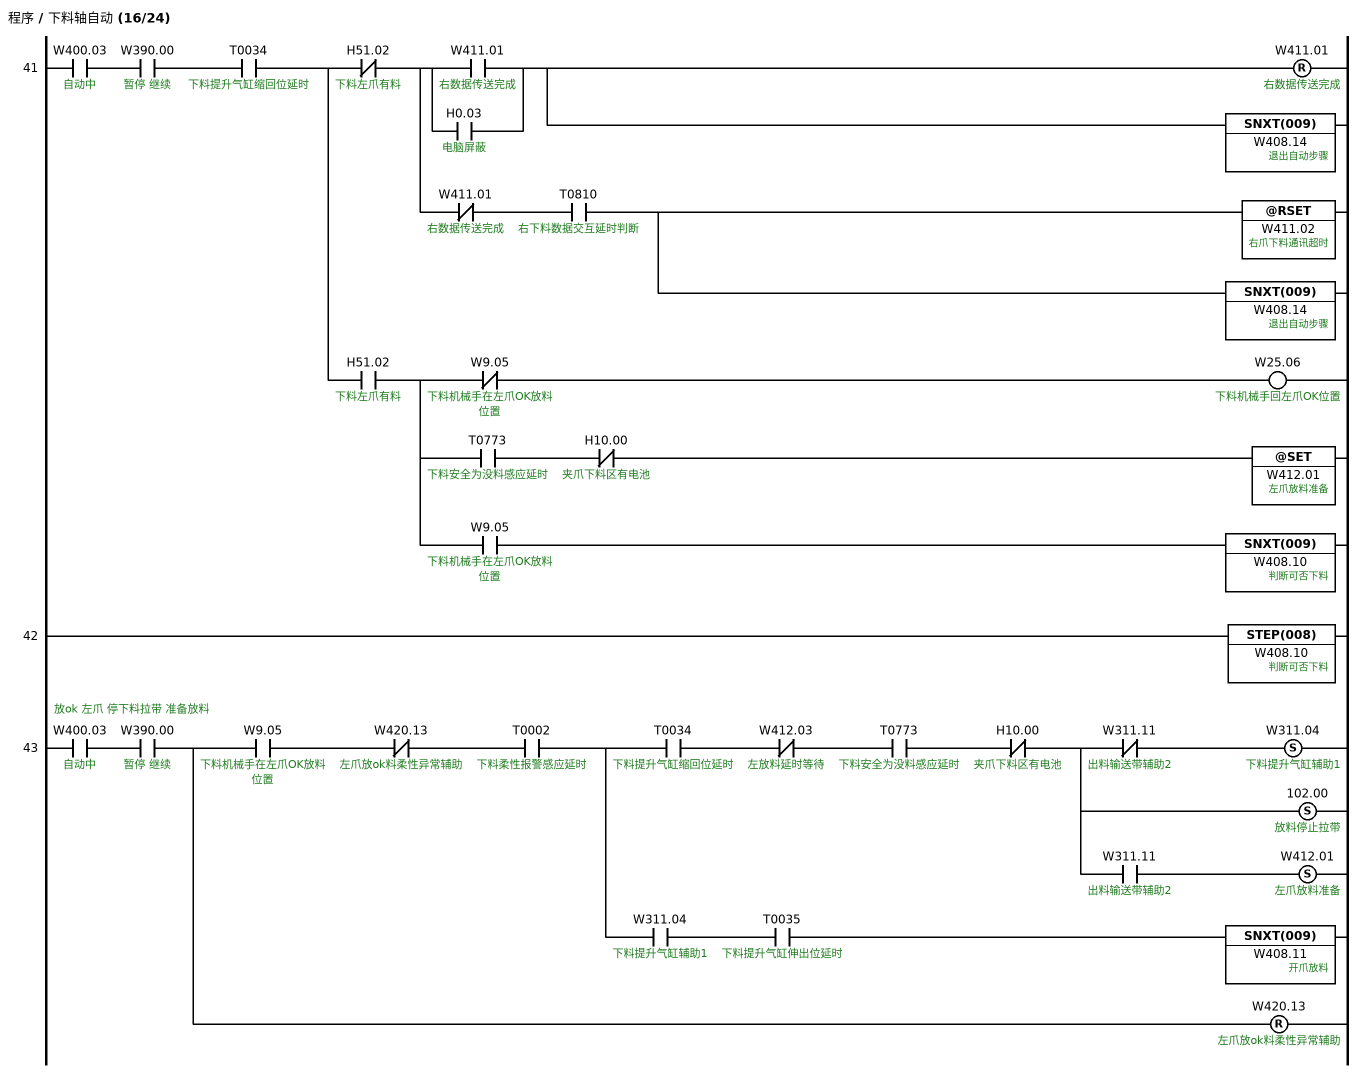
; rung 41
LD W400.03  ; 自动中
AND W390.00  ; 暂停 继续
AND T0034  ; 下料提升气缸缩回位延时
OUT TR0
ANDNOT H51.02  ; 下料左爪有料
OUT TR1
LD W411.01  ; 右数据传送完成
OR H0.03  ; 电脑屏蔽
ANDLD
RSET W411.01  ; 右数据传送完成
SNXT(009) W408.14  ; 退出自动步骤
LD TR1
ANDNOT W411.01  ; 右数据传送完成
AND T0810  ; 右下料数据交互延时判断
@RSET W411.02  ; 右爪下料通讯超时
SNXT(009) W408.14  ; 退出自动步骤
LD TR0
AND H51.02  ; 下料左爪有料
OUT TR0
ANDNOT W9.05  ; 下料机械手在左爪OK放料位置
OUT W25.06  ; 下料机械手回左爪OK位置
LD TR0
AND T0773  ; 下料安全为没料感应延时
ANDNOT H10.00  ; 夹爪下料区有电池
@SET W412.01  ; 左爪放料准备
LD TR0
AND W9.05  ; 下料机械手在左爪OK放料位置
SNXT(009) W408.10  ; 判断可否下料
; rung 42
STEP(008) W408.10  ; 判断可否下料
; rung 43: 放ok 左爪 停下料拉带 准备放料
LD W400.03  ; 自动中
AND W390.00  ; 暂停 继续
OUT TR0
AND W9.05  ; 下料机械手在左爪OK放料位置
ANDNOT W420.13  ; 左爪放ok料柔性异常辅助
AND T0002  ; 下料柔性报警感应延时
OUT TR1
AND T0034  ; 下料提升气缸缩回位延时
ANDNOT W412.03  ; 左放料延时等待
AND T0773  ; 下料安全为没料感应延时
ANDNOT H10.00  ; 夹爪下料区有电池
OUT TR2
ANDNOT W311.11  ; 出料输送带辅助2
SET W311.04  ; 下料提升气缸辅助1
LD TR2
SET 102.00  ; 放料停止拉带
AND W311.11  ; 出料输送带辅助2
SET W412.01  ; 左爪放料准备
LD TR1
AND W311.04  ; 下料提升气缸辅助1
AND T0035  ; 下料提升气缸伸出位延时
SNXT(009) W408.11  ; 开爪放料
LD TR0
RSET W420.13  ; 左爪放ok料柔性异常辅助

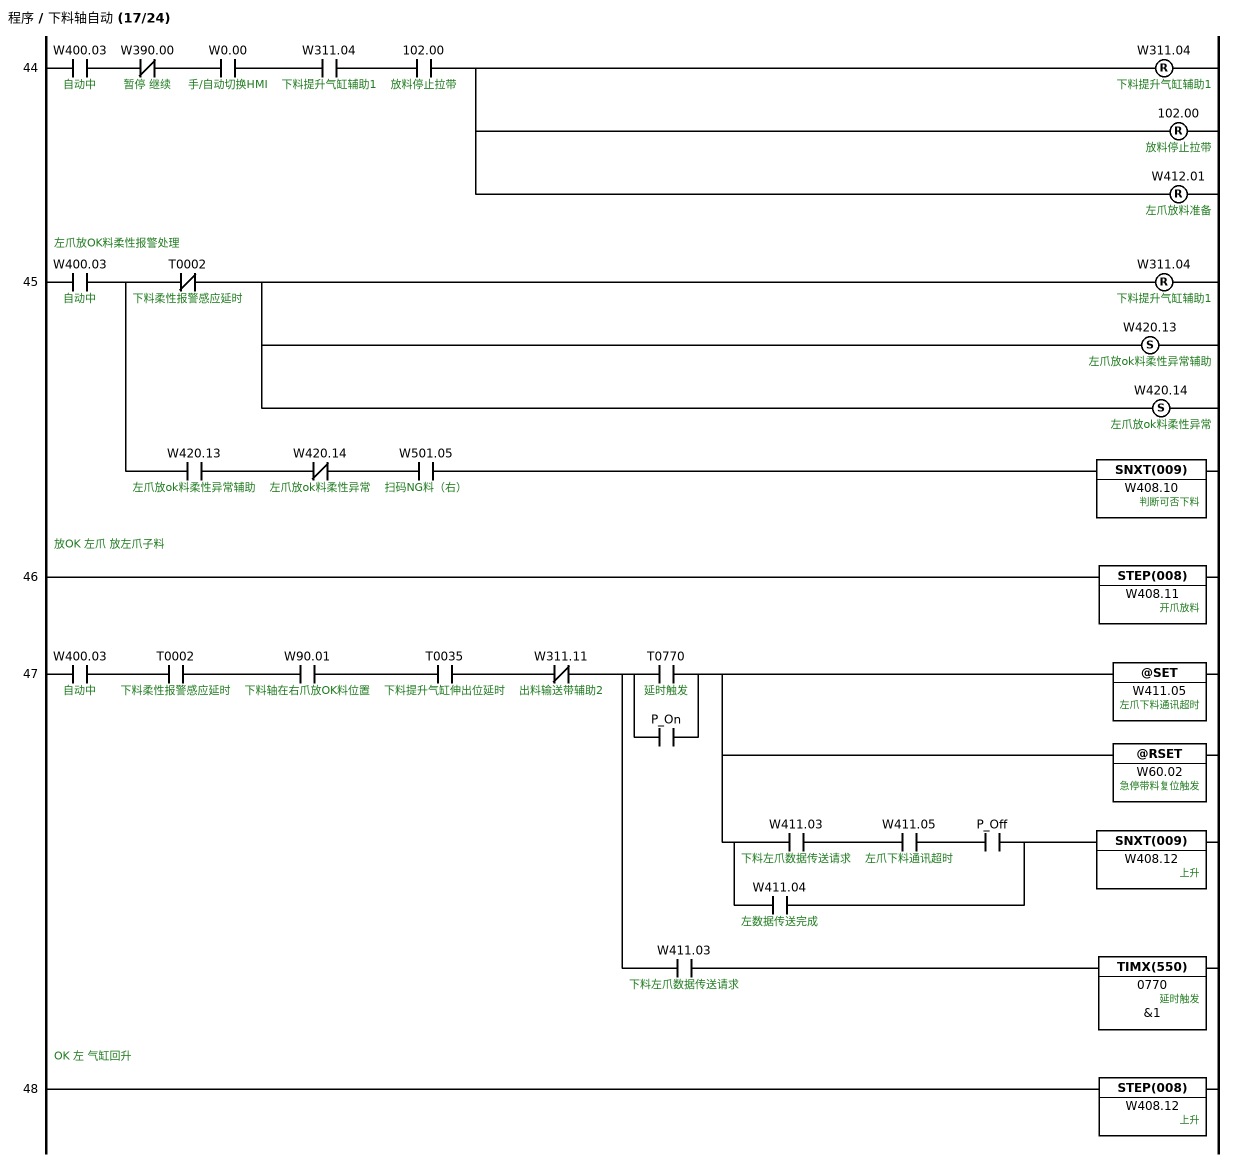
; rung 44
LD W400.03  ; 自动中
ANDNOT W390.00  ; 暂停 继续
AND W0.00  ; 手/自动切换HMI
AND W311.04  ; 下料提升气缸辅助1
AND 102.00  ; 放料停止拉带
RSET W311.04  ; 下料提升气缸辅助1
RSET 102.00  ; 放料停止拉带
RSET W412.01  ; 左爪放料准备
; rung 45: 左爪放OK料柔性报警处理
LD W400.03  ; 自动中
OUT TR0
ANDNOT T0002  ; 下料柔性报警感应延时
RSET W311.04  ; 下料提升气缸辅助1
SET W420.13  ; 左爪放ok料柔性异常辅助
SET W420.14  ; 左爪放ok料柔性异常
LD TR0
AND W420.13  ; 左爪放ok料柔性异常辅助
ANDNOT W420.14  ; 左爪放ok料柔性异常
AND W501.05  ; 扫码NG料（右）
SNXT(009) W408.10  ; 判断可否下料
; rung 46: 放OK 左爪 放左爪子料
STEP(008) W408.11  ; 开爪放料
; rung 47
LD W400.03  ; 自动中
AND T0002  ; 下料柔性报警感应延时
AND W90.01  ; 下料轴在右爪放OK料位置
AND T0035  ; 下料提升气缸伸出位延时
ANDNOT W311.11  ; 出料输送带辅助2
OUT TR0
LD T0770  ; 延时触发
OR P_On
ANDLD
@SET W411.05  ; 左爪下料通讯超时
@RSET W60.02  ; 急停带料复位触发
LD W411.03  ; 下料左爪数据传送请求
AND W411.05  ; 左爪下料通讯超时
AND P_Off
OR W411.04  ; 左数据传送完成
ANDLD
SNXT(009) W408.12  ; 上升
LD TR0
AND W411.03  ; 下料左爪数据传送请求
TIMX(550) 0770 &1  ; 延时触发
; rung 48: OK 左 气缸回升
STEP(008) W408.12  ; 上升

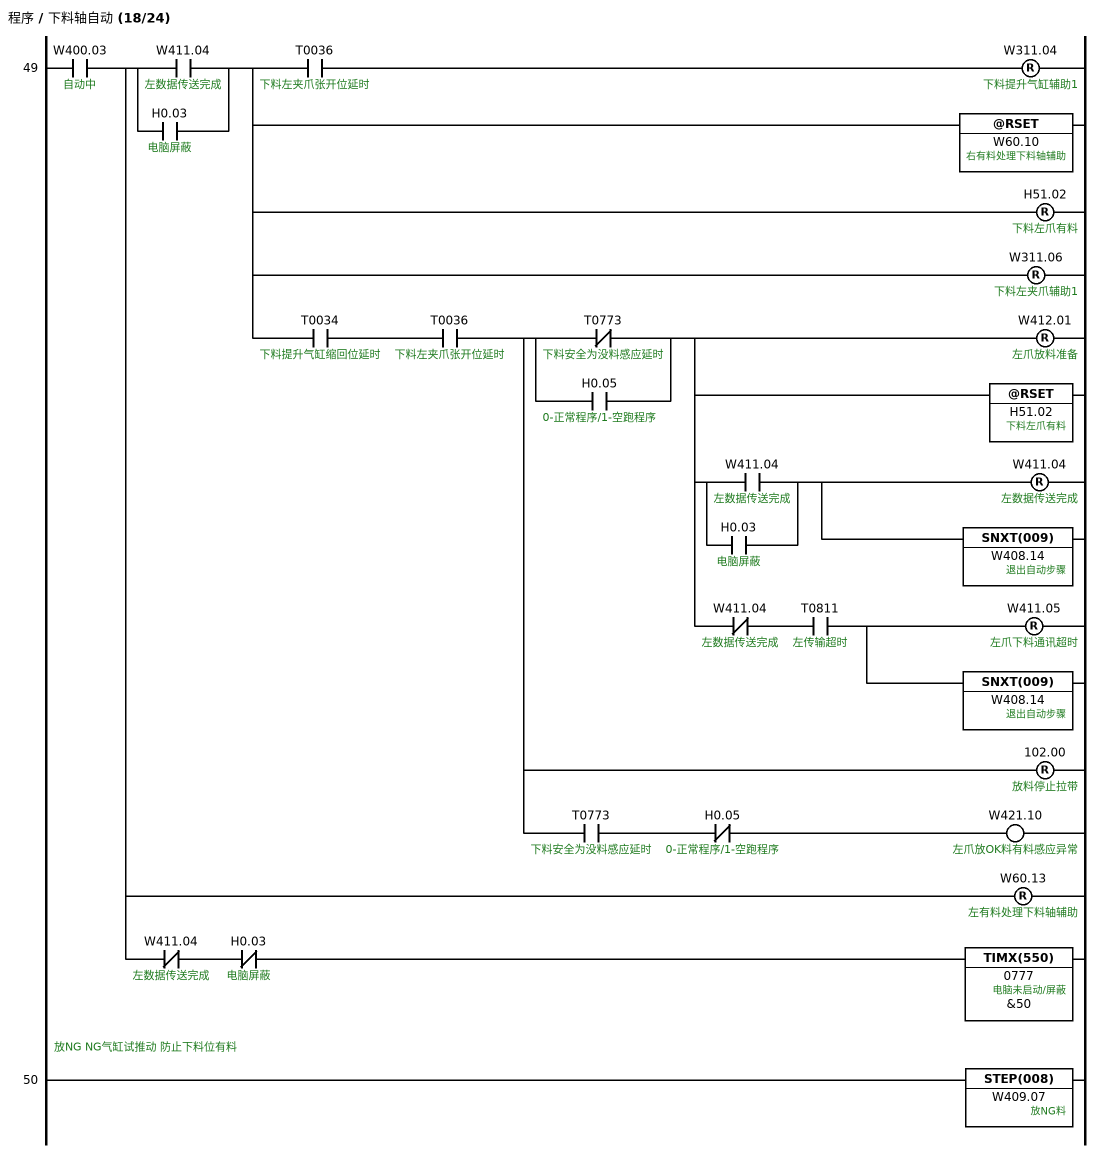
; rung 49
LD W400.03  ; 自动中
OUT TR0
LD W411.04  ; 左数据传送完成
OR H0.03  ; 电脑屏蔽
ANDLD
OUT TR1
AND T0036  ; 下料左夹爪张开位延时
RSET W311.04  ; 下料提升气缸辅助1
LD TR1
@RSET W60.10  ; 右有料处理下料轴辅助
RSET H51.02  ; 下料左爪有料
RSET W311.06  ; 下料左夹爪辅助1
AND T0034  ; 下料提升气缸缩回位延时
AND T0036  ; 下料左夹爪张开位延时
OUT TR1
LDNOT T0773  ; 下料安全为没料感应延时
OR H0.05  ; 0-正常程序/1-空跑程序
ANDLD
OUT TR2
RSET W412.01  ; 左爪放料准备
@RSET H51.02  ; 下料左爪有料
LD W411.04  ; 左数据传送完成
OR H0.03  ; 电脑屏蔽
ANDLD
RSET W411.04  ; 左数据传送完成
SNXT(009) W408.14  ; 退出自动步骤
LD TR2
ANDNOT W411.04  ; 左数据传送完成
AND T0811  ; 左传输超时
RSET W411.05  ; 左爪下料通讯超时
SNXT(009) W408.14  ; 退出自动步骤
LD TR1
RSET 102.00  ; 放料停止拉带
AND T0773  ; 下料安全为没料感应延时
ANDNOT H0.05  ; 0-正常程序/1-空跑程序
OUT W421.10  ; 左爪放OK料有料感应异常
LD TR0
RSET W60.13  ; 左有料处理下料轴辅助
ANDNOT W411.04  ; 左数据传送完成
ANDNOT H0.03  ; 电脑屏蔽
TIMX(550) 0777 &50  ; 电脑未启动/屏蔽
; rung 50: 放NG NG气缸试推动 防止下料位有料
STEP(008) W409.07  ; 放NG料

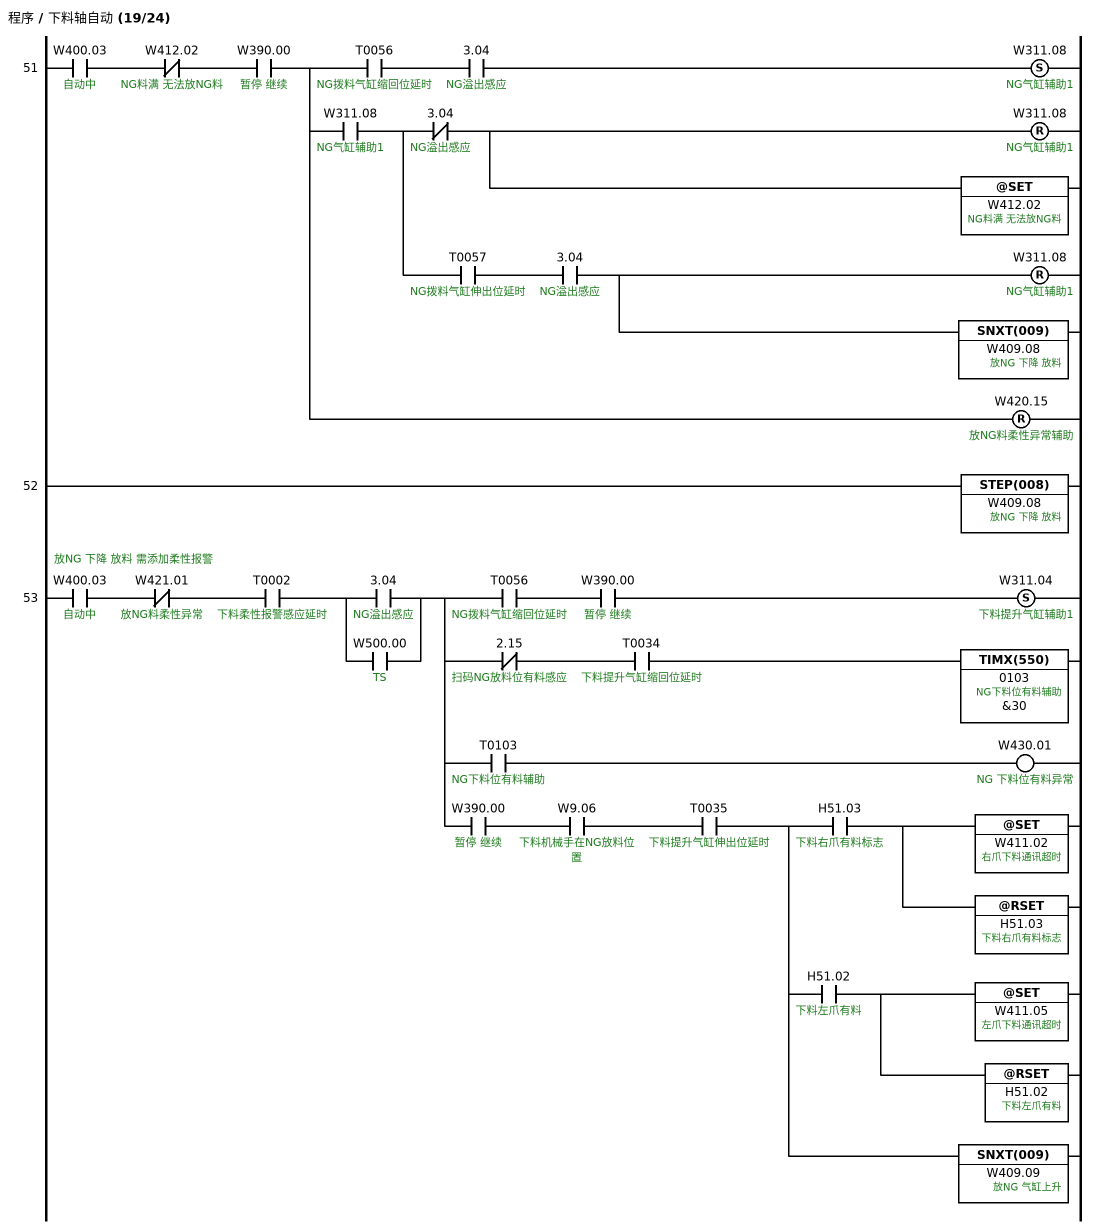
; rung 51
LD W400.03  ; 自动中
ANDNOT W412.02  ; NG料满 无法放NG料
AND W390.00  ; 暂停 继续
OUT TR0
AND T0056  ; NG拨料气缸缩回位延时
AND 3.04  ; NG溢出感应
SET W311.08  ; NG气缸辅助1
LD TR0
AND W311.08  ; NG气缸辅助1
OUT TR1
ANDNOT 3.04  ; NG溢出感应
RSET W311.08  ; NG气缸辅助1
@SET W412.02  ; NG料满 无法放NG料
LD TR1
AND T0057  ; NG拨料气缸伸出位延时
AND 3.04  ; NG溢出感应
RSET W311.08  ; NG气缸辅助1
SNXT(009) W409.08  ; 放NG 下降 放料
LD TR0
RSET W420.15  ; 放NG料柔性异常辅助
; rung 52
STEP(008) W409.08  ; 放NG 下降 放料
; rung 53: 放NG 下降 放料 需添加柔性报警
LD W400.03  ; 自动中
ANDNOT W421.01  ; 放NG料柔性异常
AND T0002  ; 下料柔性报警感应延时
LD 3.04  ; NG溢出感应
OR W500.00  ; TS
ANDLD
OUT TR0
AND T0056  ; NG拨料气缸缩回位延时
AND W390.00  ; 暂停 继续
SET W311.04  ; 下料提升气缸辅助1
LD TR0
ANDNOT 2.15  ; 扫码NG放料位有料感应
AND T0034  ; 下料提升气缸缩回位延时
TIMX(550) 0103 &30  ; NG下料位有料辅助
LD TR0
AND T0103  ; NG下料位有料辅助
OUT W430.01  ; NG 下料位有料异常
LD TR0
AND W390.00  ; 暂停 继续
AND W9.06  ; 下料机械手在NG放料位置
AND T0035  ; 下料提升气缸伸出位延时
OUT TR0
AND H51.03  ; 下料右爪有料标志
@SET W411.02  ; 右爪下料通讯超时
@RSET H51.03  ; 下料右爪有料标志
LD TR0
AND H51.02  ; 下料左爪有料
@SET W411.05  ; 左爪下料通讯超时
@RSET H51.02  ; 下料左爪有料
LD TR0
SNXT(009) W409.09  ; 放NG 气缸上升

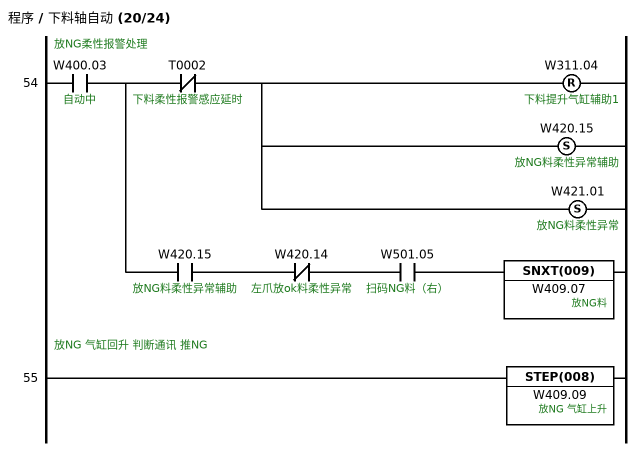
; rung 54: 放NG柔性报警处理
LD W400.03  ; 自动中
OUT TR0
ANDNOT T0002  ; 下料柔性报警感应延时
RSET W311.04  ; 下料提升气缸辅助1
SET W420.15  ; 放NG料柔性异常辅助
SET W421.01  ; 放NG料柔性异常
LD TR0
AND W420.15  ; 放NG料柔性异常辅助
ANDNOT W420.14  ; 左爪放ok料柔性异常
AND W501.05  ; 扫码NG料（右）
SNXT(009) W409.07  ; 放NG料
; rung 55: 放NG 气缸回升 判断通讯 推NG
STEP(008) W409.09  ; 放NG 气缸上升

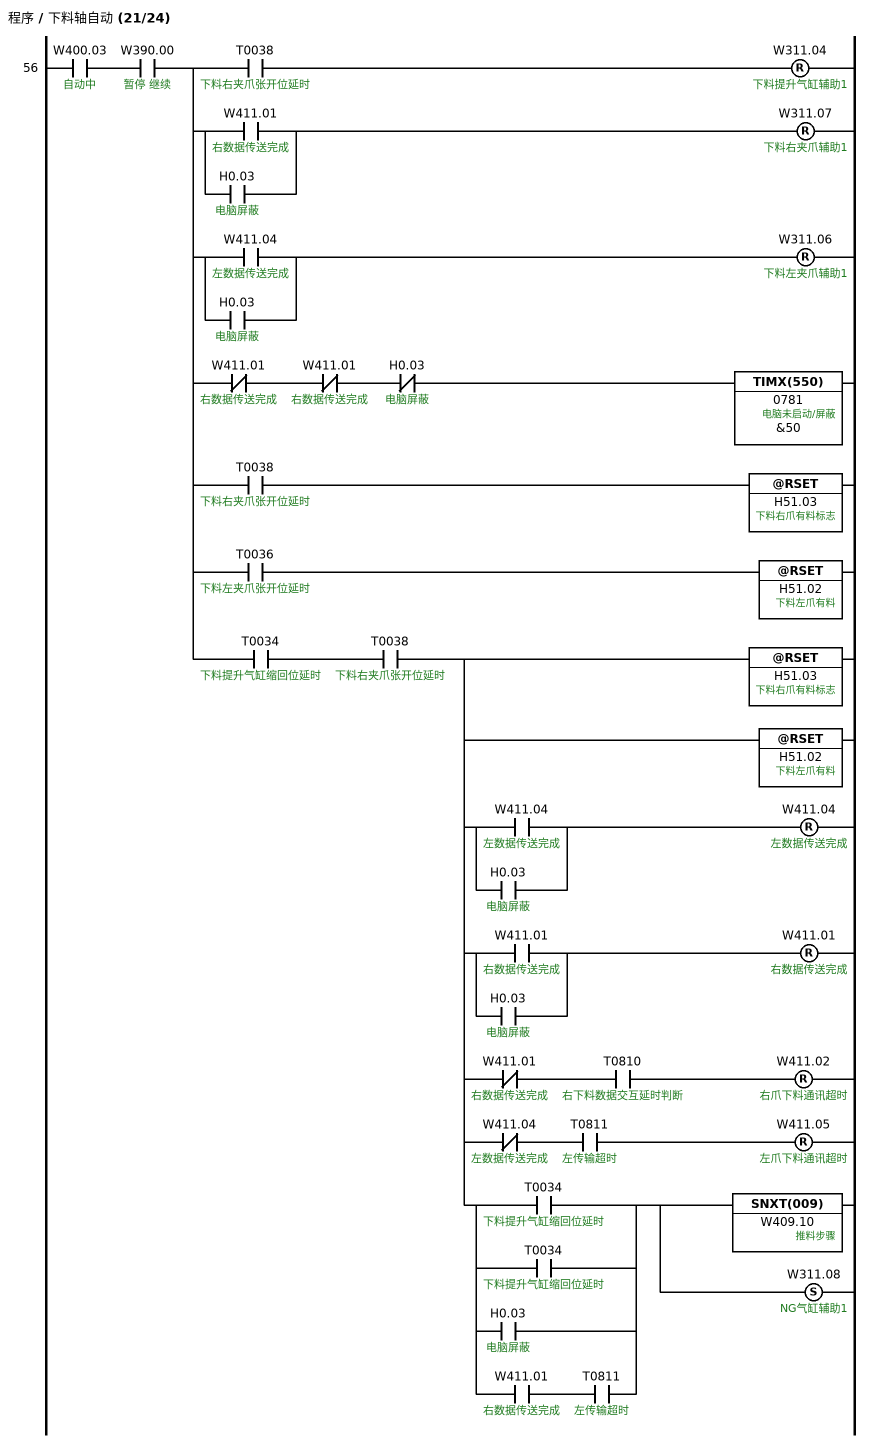
; rung 56
LD W400.03  ; 自动中
AND W390.00  ; 暂停 继续
OUT TR0
AND T0038  ; 下料右夹爪张开位延时
RSET W311.04  ; 下料提升气缸辅助1
LD TR0
LD W411.01  ; 右数据传送完成
OR H0.03  ; 电脑屏蔽
ANDLD
RSET W311.07  ; 下料右夹爪辅助1
LD TR0
LD W411.04  ; 左数据传送完成
OR H0.03  ; 电脑屏蔽
ANDLD
RSET W311.06  ; 下料左夹爪辅助1
LD TR0
ANDNOT W411.01  ; 右数据传送完成
ANDNOT W411.01  ; 右数据传送完成
ANDNOT H0.03  ; 电脑屏蔽
TIMX(550) 0781 &50  ; 电脑未启动/屏蔽
LD TR0
AND T0038  ; 下料右夹爪张开位延时
@RSET H51.03  ; 下料右爪有料标志
LD TR0
AND T0036  ; 下料左夹爪张开位延时
@RSET H51.02  ; 下料左爪有料
LD TR0
AND T0034  ; 下料提升气缸缩回位延时
AND T0038  ; 下料右夹爪张开位延时
OUT TR0
@RSET H51.03  ; 下料右爪有料标志
@RSET H51.02  ; 下料左爪有料
LD W411.04  ; 左数据传送完成
OR H0.03  ; 电脑屏蔽
ANDLD
RSET W411.04  ; 左数据传送完成
LD TR0
LD W411.01  ; 右数据传送完成
OR H0.03  ; 电脑屏蔽
ANDLD
RSET W411.01  ; 右数据传送完成
LD TR0
ANDNOT W411.01  ; 右数据传送完成
AND T0810  ; 右下料数据交互延时判断
RSET W411.02  ; 右爪下料通讯超时
LD TR0
ANDNOT W411.04  ; 左数据传送完成
AND T0811  ; 左传输超时
RSET W411.05  ; 左爪下料通讯超时
LD TR0
LD T0034  ; 下料提升气缸缩回位延时
OR T0034  ; 下料提升气缸缩回位延时
OR H0.03  ; 电脑屏蔽
LD W411.01  ; 右数据传送完成
AND T0811  ; 左传输超时
ORLD
ANDLD
SNXT(009) W409.10  ; 推料步骤
SET W311.08  ; NG气缸辅助1

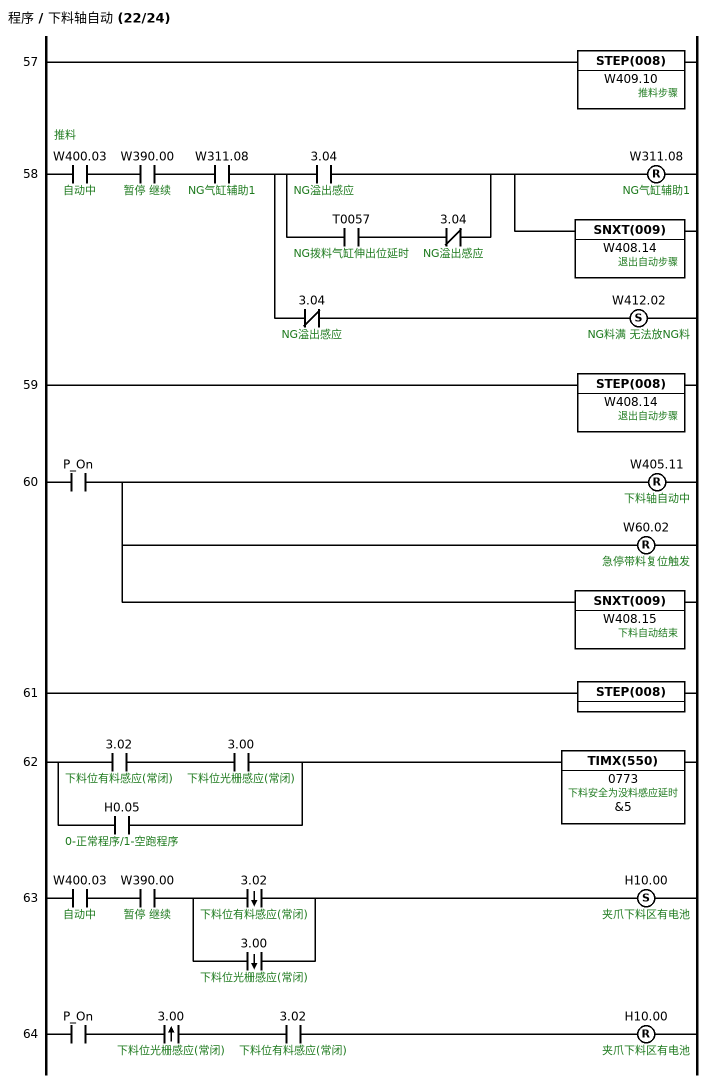
; rung 57
STEP(008) W409.10  ; 推料步骤
; rung 58: 推料
LD W400.03  ; 自动中
AND W390.00  ; 暂停 继续
AND W311.08  ; NG气缸辅助1
OUT TR0
LD 3.04  ; NG溢出感应
LD T0057  ; NG拨料气缸伸出位延时
ANDNOT 3.04  ; NG溢出感应
ORLD
ANDLD
RSET W311.08  ; NG气缸辅助1
SNXT(009) W408.14  ; 退出自动步骤
LD TR0
ANDNOT 3.04  ; NG溢出感应
SET W412.02  ; NG料满 无法放NG料
; rung 59
STEP(008) W408.14  ; 退出自动步骤
; rung 60
LD P_On
RSET W405.11  ; 下料轴自动中
RSET W60.02  ; 急停带料复位触发
SNXT(009) W408.15  ; 下料自动结束
; rung 61
STEP(008)
; rung 62
LD 3.02  ; 下料位有料感应(常闭)
AND 3.00  ; 下料位光栅感应(常闭)
OR H0.05  ; 0-正常程序/1-空跑程序
TIMX(550) 0773 &5  ; 下料安全为没料感应延时
; rung 63
LD W400.03  ; 自动中
AND W390.00  ; 暂停 继续
%LD 3.02  ; 下料位有料感应(常闭)
%OR 3.00  ; 下料位光栅感应(常闭)
ANDLD
SET H10.00  ; 夹爪下料区有电池
; rung 64
LD P_On
@AND 3.00  ; 下料位光栅感应(常闭)
AND 3.02  ; 下料位有料感应(常闭)
RSET H10.00  ; 夹爪下料区有电池

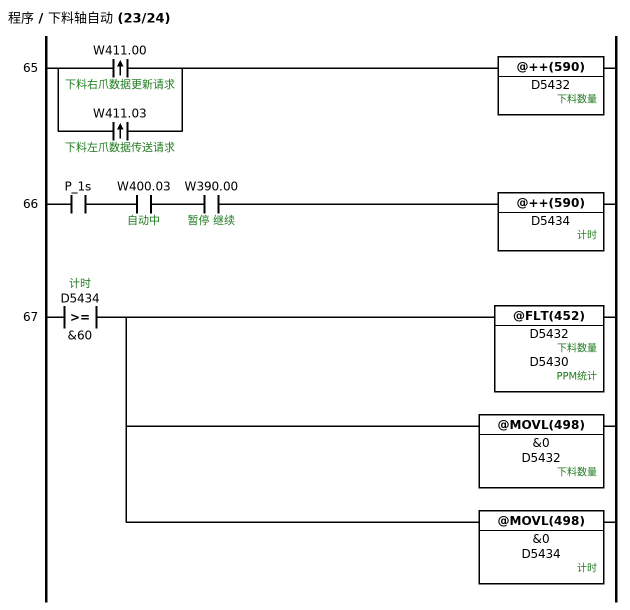
; rung 65
@LD W411.00  ; 下料右爪数据更新请求
@OR W411.03  ; 下料左爪数据传送请求
@++(590) D5432  ; 下料数量
; rung 66
LD P_1s
AND W400.03  ; 自动中
AND W390.00  ; 暂停 继续
@++(590) D5434  ; 计时
; rung 67
LD>=(325) D5434 &60  ; 计时
@FLT(452) D5432 D5430  ; 下料数量, PPM统计
@MOVL(498) &0 D5432  ; 下料数量
@MOVL(498) &0 D5434  ; 计时

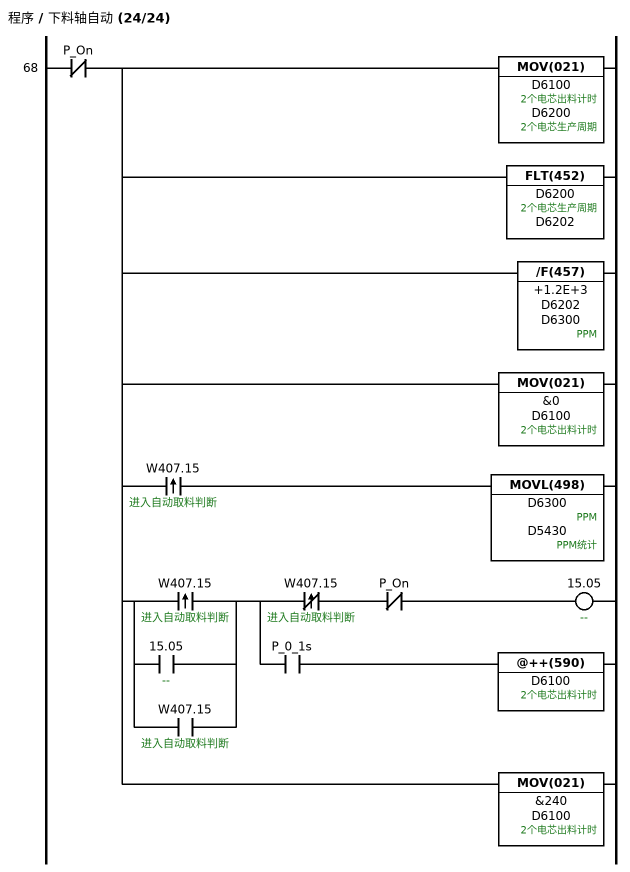
; rung 68
LDNOT P_On
OUT TR0
MOV(021) D6100 D6200  ; 2个电芯出料计时, 2个电芯生产周期
FLT(452) D6200 D6202  ; 2个电芯生产周期
/F(457) +1.2E+3 D6202 D6300  ; PPM
MOV(021) &0 D6100  ; 2个电芯出料计时
@AND W407.15  ; 进入自动取料判断
MOVL(498) D6300 D5430  ; PPM, PPM统计
LD TR0
@LD W407.15  ; 进入自动取料判断
OR 15.05  ; --
OR W407.15  ; 进入自动取料判断
ANDLD
OUT TR1
@ANDNOT W407.15  ; 进入自动取料判断
ANDNOT P_On
OUT 15.05  ; --
LD TR1
AND P_0_1s
@++(590) D6100  ; 2个电芯出料计时
LD TR0
MOV(021) &240 D6100  ; 2个电芯出料计时

### Section PC交换

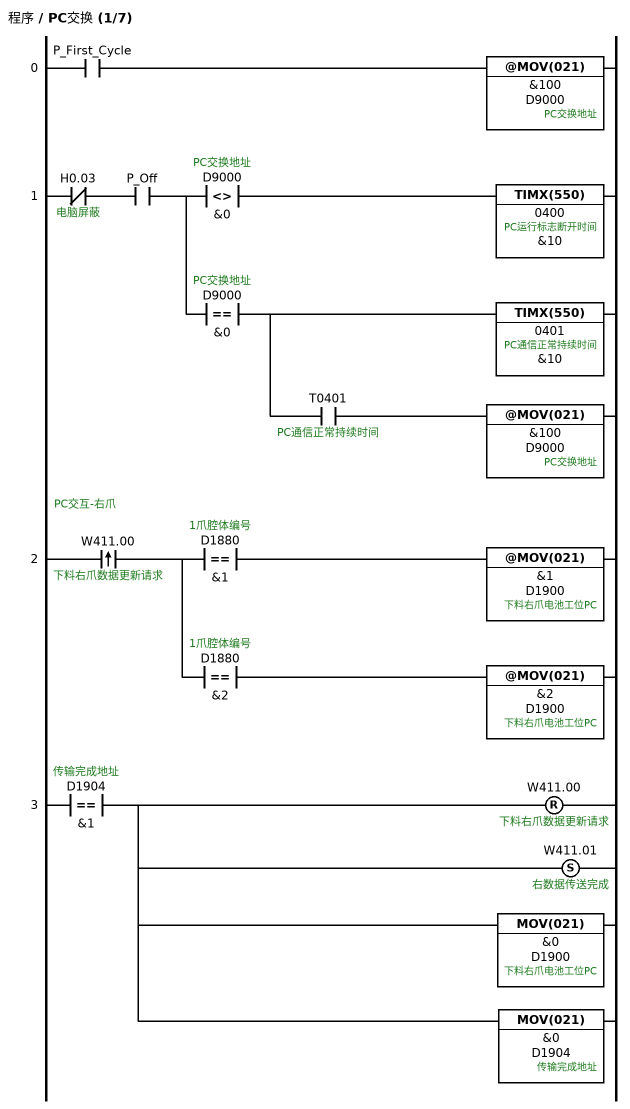
; rung 0
LD P_First_Cycle
@MOV(021) &100 D9000  ; PC交换地址
; rung 1
LDNOT H0.03  ; 电脑屏蔽
AND P_Off
OUT TR0
AND<>(305) D9000 &0  ; PC交换地址
TIMX(550) 0400 &10  ; PC运行标志断开时间
LD TR0
AND=(300) D9000 &0  ; PC交换地址
TIMX(550) 0401 &10  ; PC通信正常持续时间
AND T0401  ; PC通信正常持续时间
@MOV(021) &100 D9000  ; PC交换地址
; rung 2: PC交互-右爪
@LD W411.00  ; 下料右爪数据更新请求
OUT TR0
AND=(300) D1880 &1  ; 1爪腔体编号
@MOV(021) &1 D1900  ; 下料右爪电池工位PC
LD TR0
AND=(300) D1880 &2  ; 1爪腔体编号
@MOV(021) &2 D1900  ; 下料右爪电池工位PC
; rung 3
LD=(300) D1904 &1  ; 传输完成地址
RSET W411.00  ; 下料右爪数据更新请求
SET W411.01  ; 右数据传送完成
MOV(021) &0 D1900  ; 下料右爪电池工位PC
MOV(021) &0 D1904  ; 传输完成地址

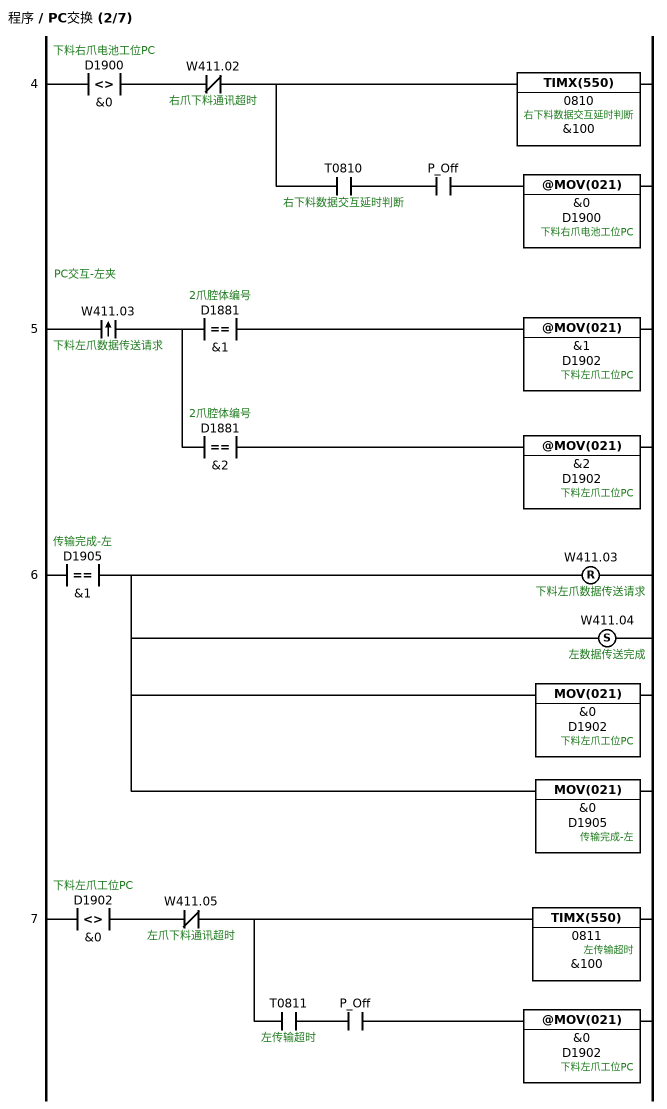
; rung 4
LD<>(305) D1900 &0  ; 下料右爪电池工位PC
ANDNOT W411.02  ; 右爪下料通讯超时
TIMX(550) 0810 &100  ; 右下料数据交互延时判断
AND T0810  ; 右下料数据交互延时判断
AND P_Off
@MOV(021) &0 D1900  ; 下料右爪电池工位PC
; rung 5: PC交互-左夹
@LD W411.03  ; 下料左爪数据传送请求
OUT TR0
AND=(300) D1881 &1  ; 2爪腔体编号
@MOV(021) &1 D1902  ; 下料左爪工位PC
LD TR0
AND=(300) D1881 &2  ; 2爪腔体编号
@MOV(021) &2 D1902  ; 下料左爪工位PC
; rung 6
LD=(300) D1905 &1  ; 传输完成-左
RSET W411.03  ; 下料左爪数据传送请求
SET W411.04  ; 左数据传送完成
MOV(021) &0 D1902  ; 下料左爪工位PC
MOV(021) &0 D1905  ; 传输完成-左
; rung 7
LD<>(305) D1902 &0  ; 下料左爪工位PC
ANDNOT W411.05  ; 左爪下料通讯超时
TIMX(550) 0811 &100  ; 左传输超时
AND T0811  ; 左传输超时
AND P_Off
@MOV(021) &0 D1902  ; 下料左爪工位PC

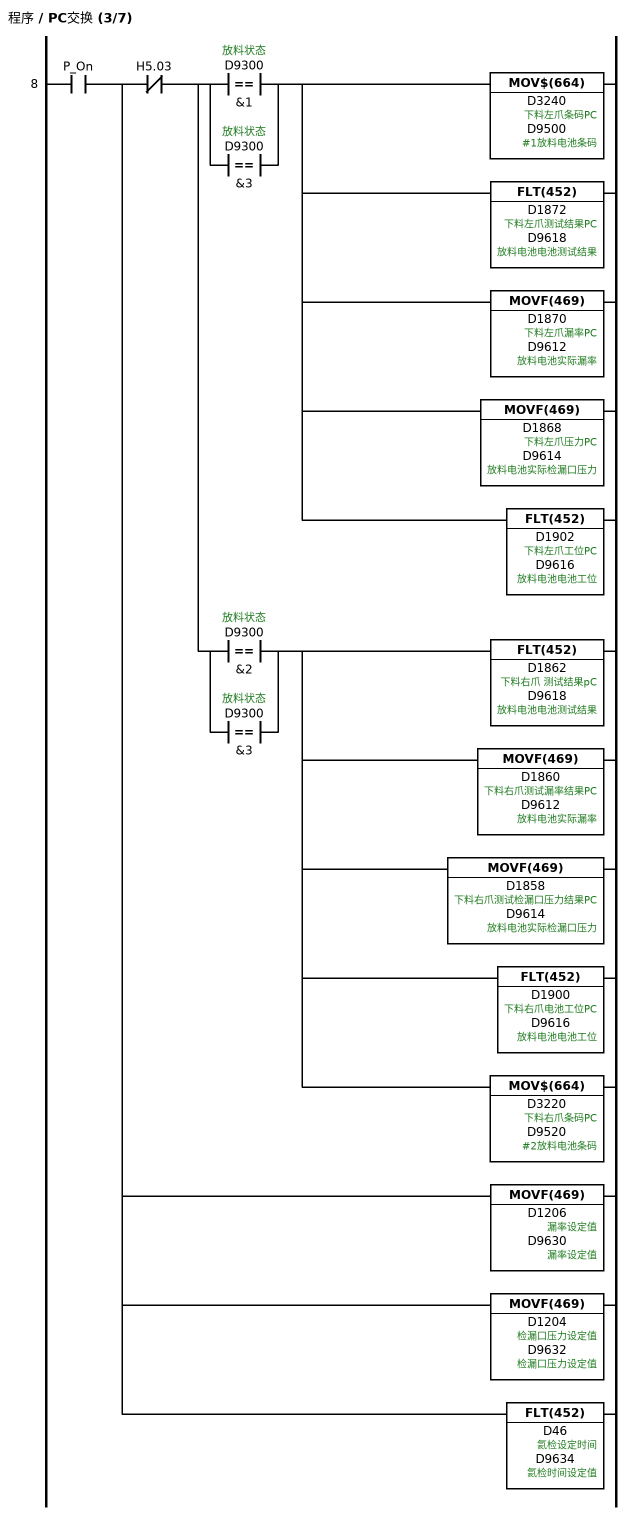
; rung 8
LD P_On
OUT TR0
ANDNOT H5.03
OUT TR1
LD=L(301) D9300 &1  ; 放料状态
OR=L(301) D9300 &3  ; 放料状态
ANDLD
MOV$(664) D3240 D9500  ; 下料左爪条码PC, #1放料电池条码
FLT(452) D1872 D9618  ; 下料左爪测试结果PC, 放料电池电池测试结果
MOVF(469) D1870 D9612  ; 下料左爪漏率PC, 放料电池实际漏率
MOVF(469) D1868 D9614  ; 下料左爪压力PC, 放料电池实际检漏口压力
FLT(452) D1902 D9616  ; 下料左爪工位PC, 放料电池电池工位
LD TR1
LD=L(301) D9300 &2  ; 放料状态
OR=L(301) D9300 &3  ; 放料状态
ANDLD
FLT(452) D1862 D9618  ; 下料右爪 测试结果pC, 放料电池电池测试结果
MOVF(469) D1860 D9612  ; 下料右爪测试漏率结果PC, 放料电池实际漏率
MOVF(469) D1858 D9614  ; 下料右爪测试检漏口压力结果PC, 放料电池实际检漏口压力
FLT(452) D1900 D9616  ; 下料右爪电池工位PC, 放料电池电池工位
MOV$(664) D3220 D9520  ; 下料右爪条码PC, #2放料电池条码
LD TR0
MOVF(469) D1206 D9630  ; 漏率设定值
MOVF(469) D1204 D9632  ; 检漏口压力设定值
FLT(452) D46 D9634  ; 氦检设定时间, 氦检时间设定值

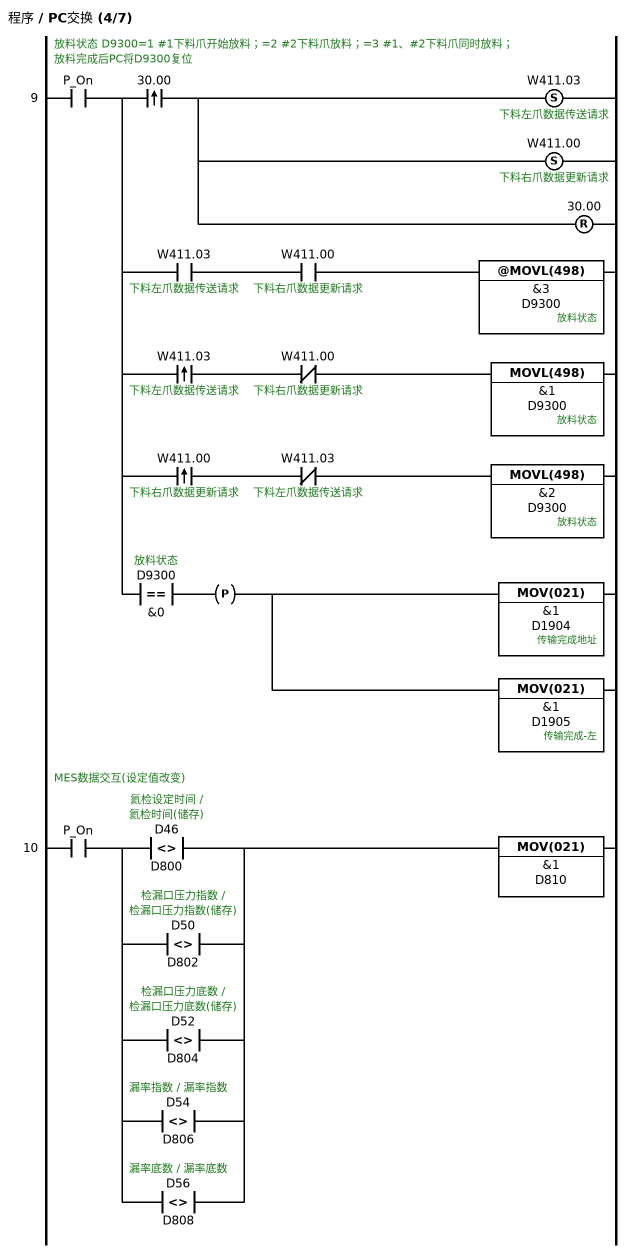
; rung 9: 放料状态 D9300=1 #1下料爪开始放料；=2 #2下料爪放料；=3 #1、#2下料爪同时放料； / 放料完成后PC将D9300复位
LD P_On
OUT TR0
@AND 30.00
SET W411.03  ; 下料左爪数据传送请求
SET W411.00  ; 下料右爪数据更新请求
RSET 30.00
LD TR0
AND W411.03  ; 下料左爪数据传送请求
AND W411.00  ; 下料右爪数据更新请求
@MOVL(498) &3 D9300  ; 放料状态
LD TR0
@AND W411.03  ; 下料左爪数据传送请求
ANDNOT W411.00  ; 下料右爪数据更新请求
MOVL(498) &1 D9300  ; 放料状态
LD TR0
@AND W411.00  ; 下料右爪数据更新请求
ANDNOT W411.03  ; 下料左爪数据传送请求
MOVL(498) &2 D9300  ; 放料状态
LD TR0
AND=L(301) D9300 &0  ; 放料状态
UP(521)
MOV(021) &1 D1904  ; 传输完成地址
MOV(021) &1 D1905  ; 传输完成-左
; rung 10: MES数据交互(设定值改变)
LD P_On
LD<>(305) D46 D800  ; 氦检设定时间, 氦检时间(储存)
OR<>F(330) D50 D802  ; 检漏口压力指数, 检漏口压力指数(储存)
OR<>F(330) D52 D804  ; 检漏口压力底数, 检漏口压力底数(储存)
OR<>F(330) D54 D806  ; 漏率指数
OR<>F(330) D56 D808  ; 漏率底数
ANDLD
MOV(021) &1 D810

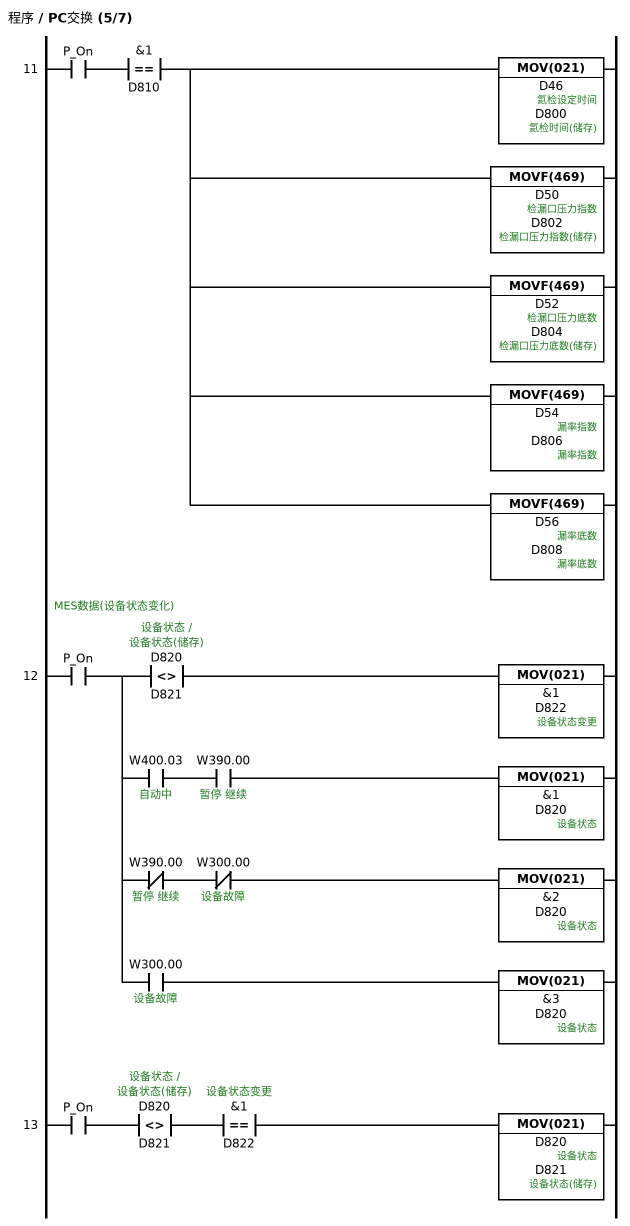
; rung 11
LD P_On
AND=(300) &1 D810
MOV(021) D46 D800  ; 氦检设定时间, 氦检时间(储存)
MOVF(469) D50 D802  ; 检漏口压力指数, 检漏口压力指数(储存)
MOVF(469) D52 D804  ; 检漏口压力底数, 检漏口压力底数(储存)
MOVF(469) D54 D806  ; 漏率指数
MOVF(469) D56 D808  ; 漏率底数
; rung 12: MES数据(设备状态变化)
LD P_On
OUT TR0
AND<>(305) D820 D821  ; 设备状态, 设备状态(储存)
MOV(021) &1 D822  ; 设备状态变更
LD TR0
AND W400.03  ; 自动中
AND W390.00  ; 暂停 继续
MOV(021) &1 D820  ; 设备状态
LD TR0
ANDNOT W390.00  ; 暂停 继续
ANDNOT W300.00  ; 设备故障
MOV(021) &2 D820  ; 设备状态
LD TR0
AND W300.00  ; 设备故障
MOV(021) &3 D820  ; 设备状态
; rung 13
LD P_On
AND<>(305) D820 D821  ; 设备状态, 设备状态(储存)
AND=(300) &1 D822  ; 设备状态变更
MOV(021) D820 D821  ; 设备状态, 设备状态(储存)

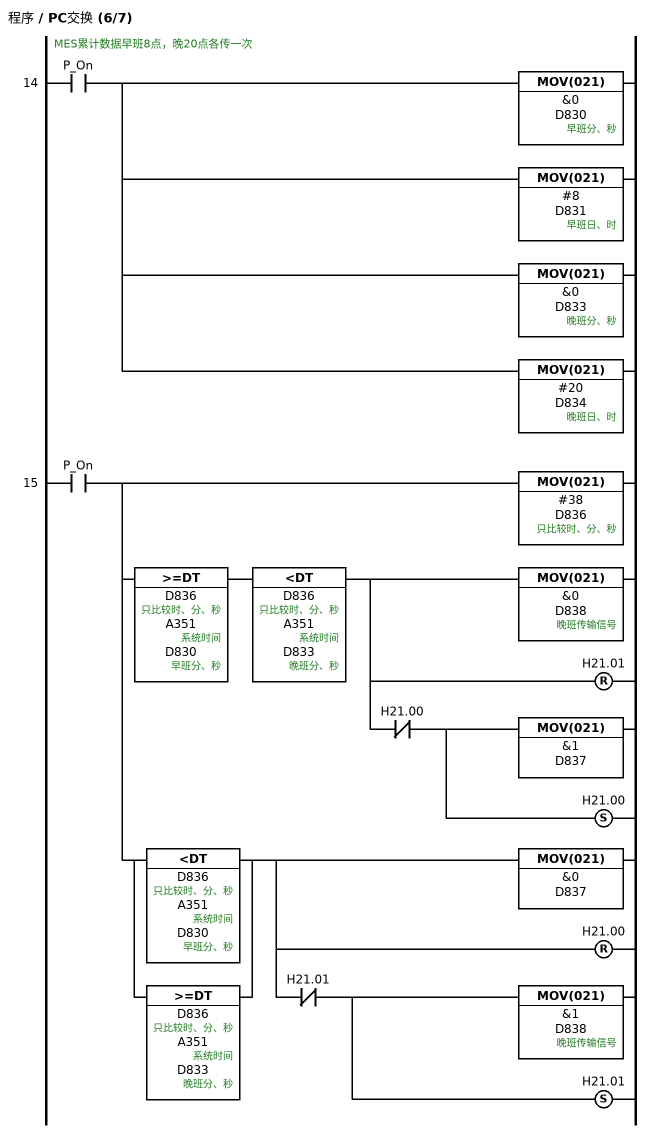
; rung 14: MES累计数据早班8点，晚20点各传一次
LD P_On
MOV(021) &0 D830  ; 早班分、秒
MOV(021) #8 D831  ; 早班日、时
MOV(021) &0 D833  ; 晚班分、秒
MOV(021) #20 D834  ; 晚班日、时
; rung 15
LD P_On
OUT TR0
MOV(021) #38 D836  ; 只比较时、分、秒
AND>=DT(346) D836 A351 D830  ; 只比较时、分、秒, 系统时间, 早班分、秒
AND<DT(343) D836 A351 D833  ; 只比较时、分、秒, 系统时间, 晚班分、秒
MOV(021) &0 D838  ; 晚班传输信号
RSET H21.01
ANDNOT H21.00
MOV(021) &1 D837
SET H21.00
LD TR0
LD<DT(343) D836 A351 D830  ; 只比较时、分、秒, 系统时间, 早班分、秒
OR>=DT(346) D836 A351 D833  ; 只比较时、分、秒, 系统时间, 晚班分、秒
ANDLD
MOV(021) &0 D837
RSET H21.00
ANDNOT H21.01
MOV(021) &1 D838  ; 晚班传输信号
SET H21.01

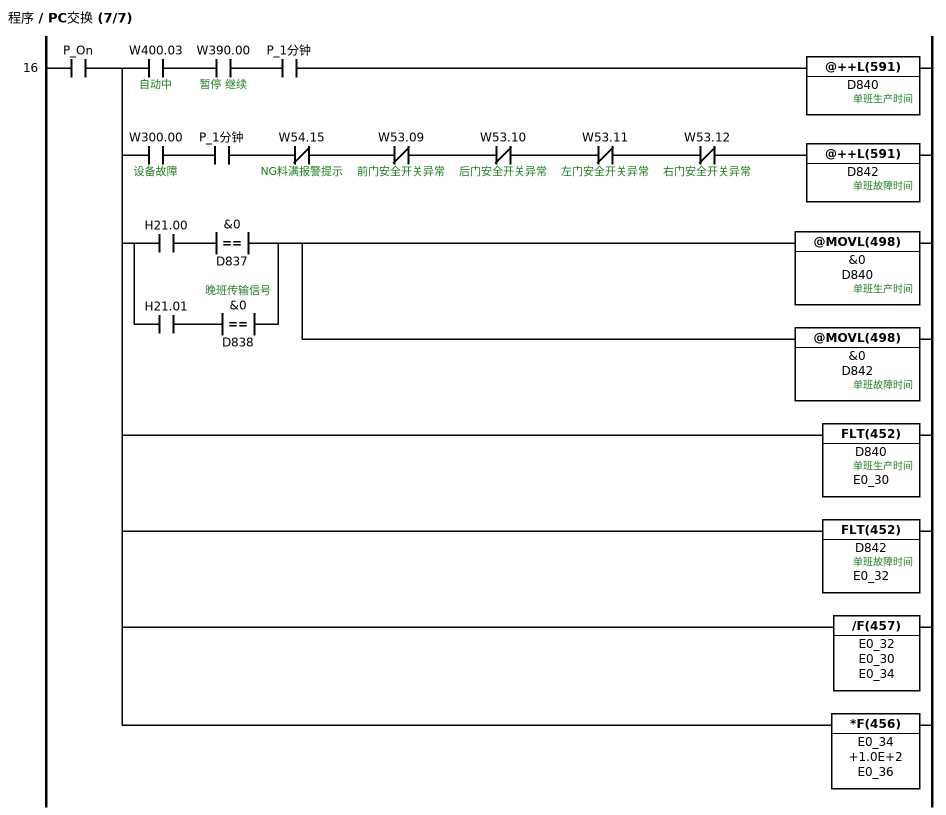
; rung 16
LD P_On
OUT TR0
AND W400.03  ; 自动中
AND W390.00  ; 暂停 继续
AND P_1分钟
@++L(591) D840  ; 单班生产时间
LD TR0
AND W300.00  ; 设备故障
AND P_1分钟
ANDNOT W54.15  ; NG料满报警提示
ANDNOT W53.09  ; 前门安全开关异常
ANDNOT W53.10  ; 后门安全开关异常
ANDNOT W53.11  ; 左门安全开关异常
ANDNOT W53.12  ; 右门安全开关异常
@++L(591) D842  ; 单班故障时间
LD TR0
LD H21.00
AND=(300) &0 D837
LD H21.01
AND=(300) &0 D838  ; 晚班传输信号
ORLD
ANDLD
@MOVL(498) &0 D840  ; 单班生产时间
@MOVL(498) &0 D842  ; 单班故障时间
LD TR0
FLT(452) D840 E0_30  ; 单班生产时间
FLT(452) D842 E0_32  ; 单班故障时间
/F(457) E0_32 E0_30 E0_34
*F(456) E0_34 +1.0E+2 E0_36

### Section 下料输送带自动

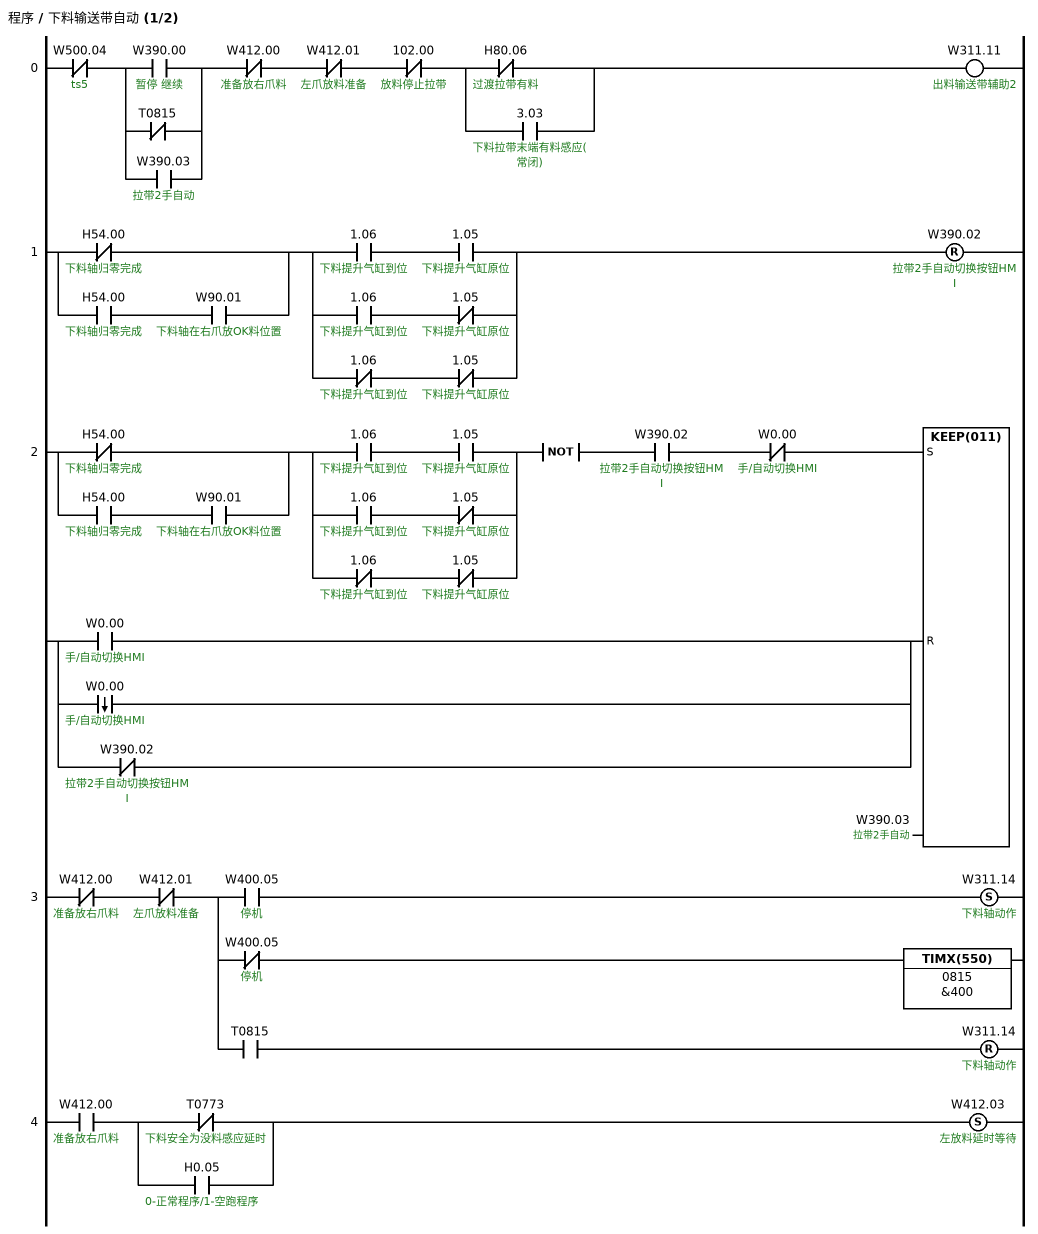
; rung 0
LDNOT W500.04  ; ts5
LD W390.00  ; 暂停 继续
ORNOT T0815
OR W390.03  ; 拉带2手自动
ANDLD
ANDNOT W412.00  ; 准备放右爪料
ANDNOT W412.01  ; 左爪放料准备
ANDNOT 102.00  ; 放料停止拉带
LDNOT H80.06  ; 过渡拉带有料
OR 3.03  ; 下料拉带末端有料感应(常闭)
ANDLD
OUT W311.11  ; 出料输送带辅助2
; rung 1
LDNOT H54.00  ; 下料轴归零完成
LD H54.00  ; 下料轴归零完成
AND W90.01  ; 下料轴在右爪放OK料位置
ORLD
LD 1.06  ; 下料提升气缸到位
AND 1.05  ; 下料提升气缸原位
LD 1.06  ; 下料提升气缸到位
ANDNOT 1.05  ; 下料提升气缸原位
ORLD
LDNOT 1.06  ; 下料提升气缸到位
ANDNOT 1.05  ; 下料提升气缸原位
ORLD
ANDLD
RSET W390.02  ; 拉带2手自动切换按钮HMI
; rung 2
LDNOT H54.00  ; 下料轴归零完成
LD H54.00  ; 下料轴归零完成
AND W90.01  ; 下料轴在右爪放OK料位置
ORLD
LD 1.06  ; 下料提升气缸到位
AND 1.05  ; 下料提升气缸原位
LD 1.06  ; 下料提升气缸到位
ANDNOT 1.05  ; 下料提升气缸原位
ORLD
LDNOT 1.06  ; 下料提升气缸到位
ANDNOT 1.05  ; 下料提升气缸原位
ORLD
ANDLD
NOT(520)
AND W390.02  ; 拉带2手自动切换按钮HMI
ANDNOT W0.00  ; 手/自动切换HMI
LD W0.00  ; 手/自动切换HMI
%OR W0.00  ; 手/自动切换HMI
ORNOT W390.02  ; 拉带2手自动切换按钮HMI
KEEP(011) W390.03  ; 拉带2手自动
; rung 3
LDNOT W412.00  ; 准备放右爪料
ANDNOT W412.01  ; 左爪放料准备
OUT TR0
AND W400.05  ; 停机
SET W311.14  ; 下料轴动作
LD TR0
ANDNOT W400.05  ; 停机
TIMX(550) 0815 &400
LD TR0
AND T0815
RSET W311.14  ; 下料轴动作
; rung 4
LD W412.00  ; 准备放右爪料
LDNOT T0773  ; 下料安全为没料感应延时
OR H0.05  ; 0-正常程序/1-空跑程序
ANDLD
SET W412.03  ; 左放料延时等待

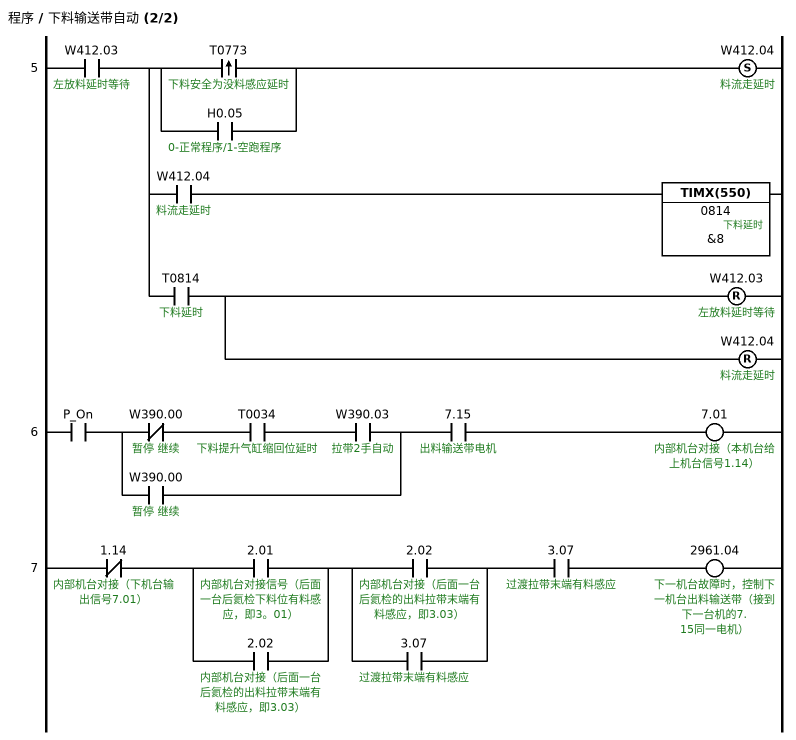
; rung 5
LD W412.03  ; 左放料延时等待
OUT TR0
@LD T0773  ; 下料安全为没料感应延时
OR H0.05  ; 0-正常程序/1-空跑程序
ANDLD
SET W412.04  ; 料流走延时
LD TR0
AND W412.04  ; 料流走延时
TIMX(550) 0814 &8  ; 下料延时
LD TR0
AND T0814  ; 下料延时
RSET W412.03  ; 左放料延时等待
RSET W412.04  ; 料流走延时
; rung 6
LD P_On
LDNOT W390.00  ; 暂停 继续
AND T0034  ; 下料提升气缸缩回位延时
AND W390.03  ; 拉带2手自动
OR W390.00  ; 暂停 继续
ANDLD
AND 7.15  ; 出料输送带电机
OUT 7.01  ; 内部机台对接（本机台给上机台信号1.14）
; rung 7
LDNOT 1.14  ; 内部机台对接（下机台输出信号7.01）
LD 2.01  ; 内部机台对接信号（后面一台后氦检下料位有料感应，即3。01）
OR 2.02  ; 内部机台对接（后面一台后氦检的出料拉带末端有料感应，即3.03）
ANDLD
LD 2.02  ; 内部机台对接（后面一台后氦检的出料拉带末端有料感应，即3.03）
OR 3.07  ; 过渡拉带末端有料感应
ANDLD
AND 3.07  ; 过渡拉带末端有料感应
OUT 2961.04  ; 下一机台故障时，控制下一机台出料输送带（接到下一台机的7.15同一电机）

### Section 气缸手动

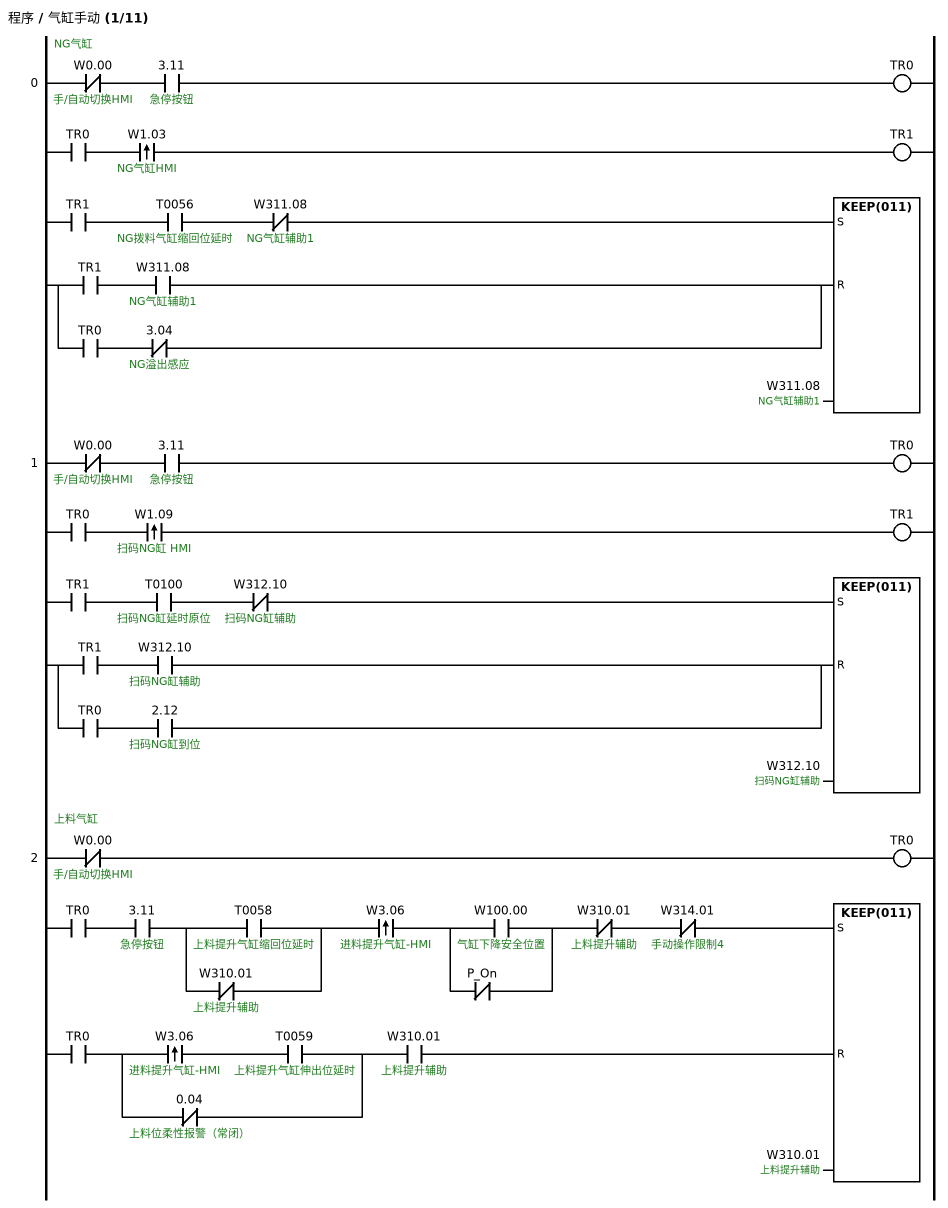
; rung 0: NG气缸
LDNOT W0.00  ; 手/自动切换HMI
AND 3.11  ; 急停按钮
OUT TR0
@AND W1.03  ; NG气缸HMI
OUT TR1
AND T0056  ; NG拨料气缸缩回位延时
ANDNOT W311.08  ; NG气缸辅助1
LD TR1
AND W311.08  ; NG气缸辅助1
LD TR0
ANDNOT 3.04  ; NG溢出感应
ORLD
KEEP(011) W311.08  ; NG气缸辅助1
; rung 1
LDNOT W0.00  ; 手/自动切换HMI
AND 3.11  ; 急停按钮
OUT TR0
@AND W1.09  ; 扫码NG缸 HMI
OUT TR1
AND T0100  ; 扫码NG缸延时原位
ANDNOT W312.10  ; 扫码NG缸辅助
LD TR1
AND W312.10  ; 扫码NG缸辅助
LD TR0
AND 2.12  ; 扫码NG缸到位
ORLD
KEEP(011) W312.10  ; 扫码NG缸辅助
; rung 2: 上料气缸
LDNOT W0.00  ; 手/自动切换HMI
OUT TR0
AND 3.11  ; 急停按钮
LD T0058  ; 上料提升气缸缩回位延时
ORNOT W310.01  ; 上料提升辅助
ANDLD
@AND W3.06  ; 进料提升气缸-HMI
LD W100.00  ; 气缸下降安全位置
ORNOT P_On
ANDLD
ANDNOT W310.01  ; 上料提升辅助
ANDNOT W314.01  ; 手动操作限制4
LD TR0
@LD W3.06  ; 进料提升气缸-HMI
AND T0059  ; 上料提升气缸伸出位延时
ORNOT 0.04  ; 上料位柔性报警（常闭）
ANDLD
AND W310.01  ; 上料提升辅助
KEEP(011) W310.01  ; 上料提升辅助

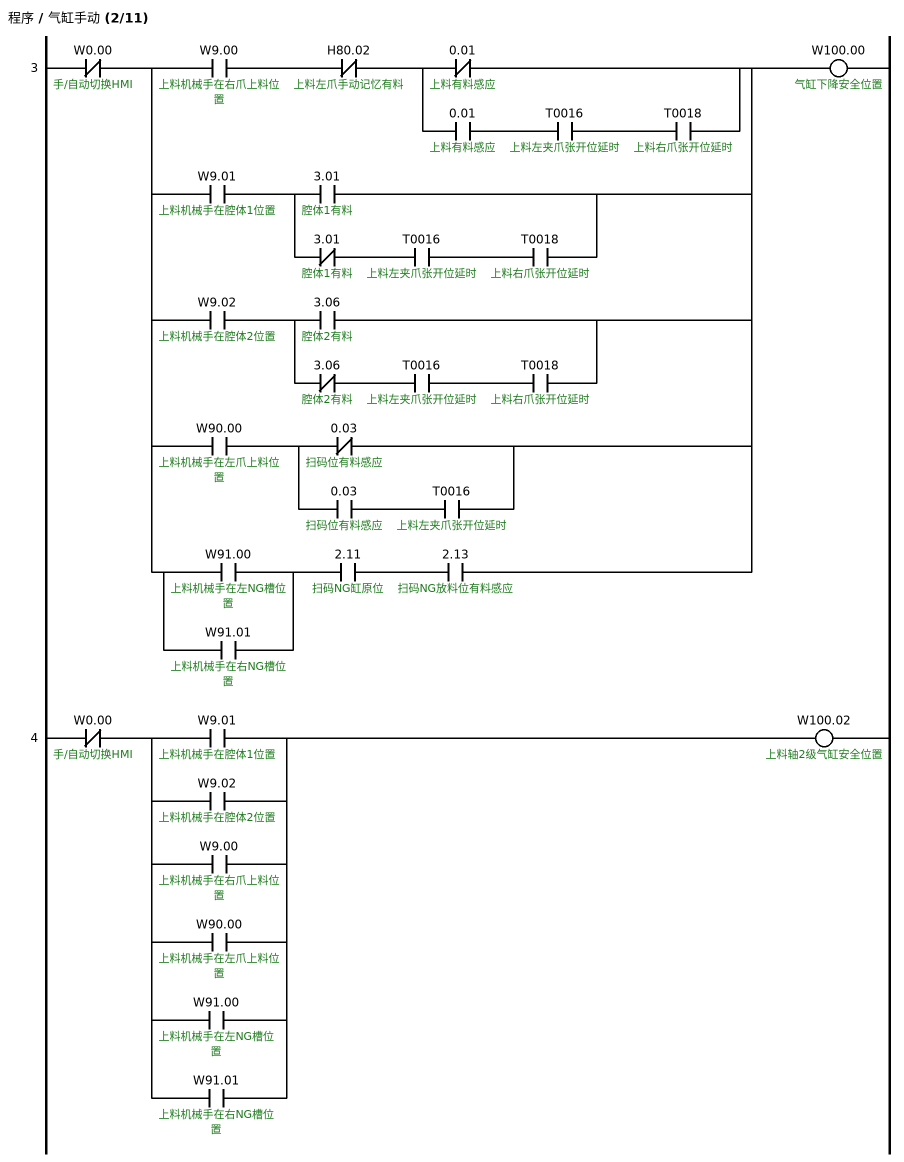
; rung 3
LDNOT W0.00  ; 手/自动切换HMI
LD W9.00  ; 上料机械手在右爪上料位置
ANDNOT H80.02  ; 上料左爪手动记忆有料
LDNOT 0.01  ; 上料有料感应
LD 0.01  ; 上料有料感应
AND T0016  ; 上料左夹爪张开位延时
AND T0018  ; 上料右爪张开位延时
ORLD
ANDLD
LD W9.01  ; 上料机械手在腔体1位置
LD 3.01  ; 腔体1有料
LDNOT 3.01  ; 腔体1有料
AND T0016  ; 上料左夹爪张开位延时
AND T0018  ; 上料右爪张开位延时
ORLD
ANDLD
ORLD
LD W9.02  ; 上料机械手在腔体2位置
LD 3.06  ; 腔体2有料
LDNOT 3.06  ; 腔体2有料
AND T0016  ; 上料左夹爪张开位延时
AND T0018  ; 上料右爪张开位延时
ORLD
ANDLD
ORLD
LD W90.00  ; 上料机械手在左爪上料位置
LDNOT 0.03  ; 扫码位有料感应
LD 0.03  ; 扫码位有料感应
AND T0016  ; 上料左夹爪张开位延时
ORLD
ANDLD
ORLD
LD W91.00  ; 上料机械手在左NG槽位置
OR W91.01  ; 上料机械手在右NG槽位置
AND 2.11  ; 扫码NG缸原位
AND 2.13  ; 扫码NG放料位有料感应
ORLD
ANDLD
OUT W100.00  ; 气缸下降安全位置
; rung 4
LDNOT W0.00  ; 手/自动切换HMI
LD W9.01  ; 上料机械手在腔体1位置
OR W9.02  ; 上料机械手在腔体2位置
OR W9.00  ; 上料机械手在右爪上料位置
OR W90.00  ; 上料机械手在左爪上料位置
OR W91.00  ; 上料机械手在左NG槽位置
OR W91.01  ; 上料机械手在右NG槽位置
ANDLD
OUT W100.02  ; 上料轴2级气缸安全位置

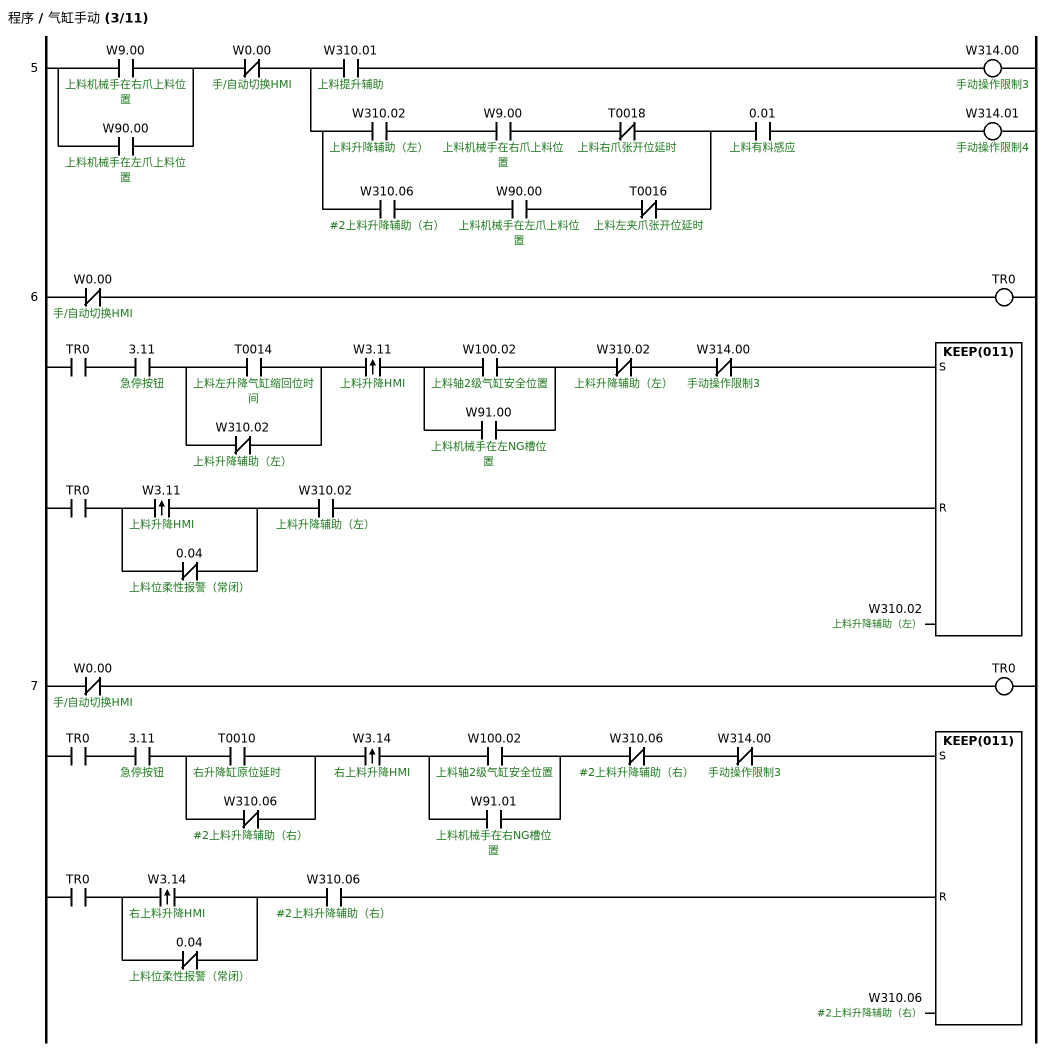
; rung 5
LD W9.00  ; 上料机械手在右爪上料位置
OR W90.00  ; 上料机械手在左爪上料位置
ANDNOT W0.00  ; 手/自动切换HMI
OUT TR0
AND W310.01  ; 上料提升辅助
OUT W314.00  ; 手动操作限制3
LD TR0
LD W310.02  ; 上料升降辅助（左）
AND W9.00  ; 上料机械手在右爪上料位置
ANDNOT T0018  ; 上料右爪张开位延时
LD W310.06  ; #2上料升降辅助（右）
AND W90.00  ; 上料机械手在左爪上料位置
ANDNOT T0016  ; 上料左夹爪张开位延时
ORLD
ANDLD
AND 0.01  ; 上料有料感应
OUT W314.01  ; 手动操作限制4
; rung 6
LDNOT W0.00  ; 手/自动切换HMI
OUT TR0
AND 3.11  ; 急停按钮
LD T0014  ; 上料左升降气缸缩回位时间
ORNOT W310.02  ; 上料升降辅助（左）
ANDLD
@AND W3.11  ; 上料升降HMI
LD W100.02  ; 上料轴2级气缸安全位置
OR W91.00  ; 上料机械手在左NG槽位置
ANDLD
ANDNOT W310.02  ; 上料升降辅助（左）
ANDNOT W314.00  ; 手动操作限制3
LD TR0
@LD W3.11  ; 上料升降HMI
ORNOT 0.04  ; 上料位柔性报警（常闭）
ANDLD
AND W310.02  ; 上料升降辅助（左）
KEEP(011) W310.02  ; 上料升降辅助（左）
; rung 7
LDNOT W0.00  ; 手/自动切换HMI
OUT TR0
AND 3.11  ; 急停按钮
LD T0010  ; 右升降缸原位延时
ORNOT W310.06  ; #2上料升降辅助（右）
ANDLD
@AND W3.14  ; 右上料升降HMI
LD W100.02  ; 上料轴2级气缸安全位置
OR W91.01  ; 上料机械手在右NG槽位置
ANDLD
ANDNOT W310.06  ; #2上料升降辅助（右）
ANDNOT W314.00  ; 手动操作限制3
LD TR0
@LD W3.14  ; 右上料升降HMI
ORNOT 0.04  ; 上料位柔性报警（常闭）
ANDLD
AND W310.06  ; #2上料升降辅助（右）
KEEP(011) W310.06  ; #2上料升降辅助（右）

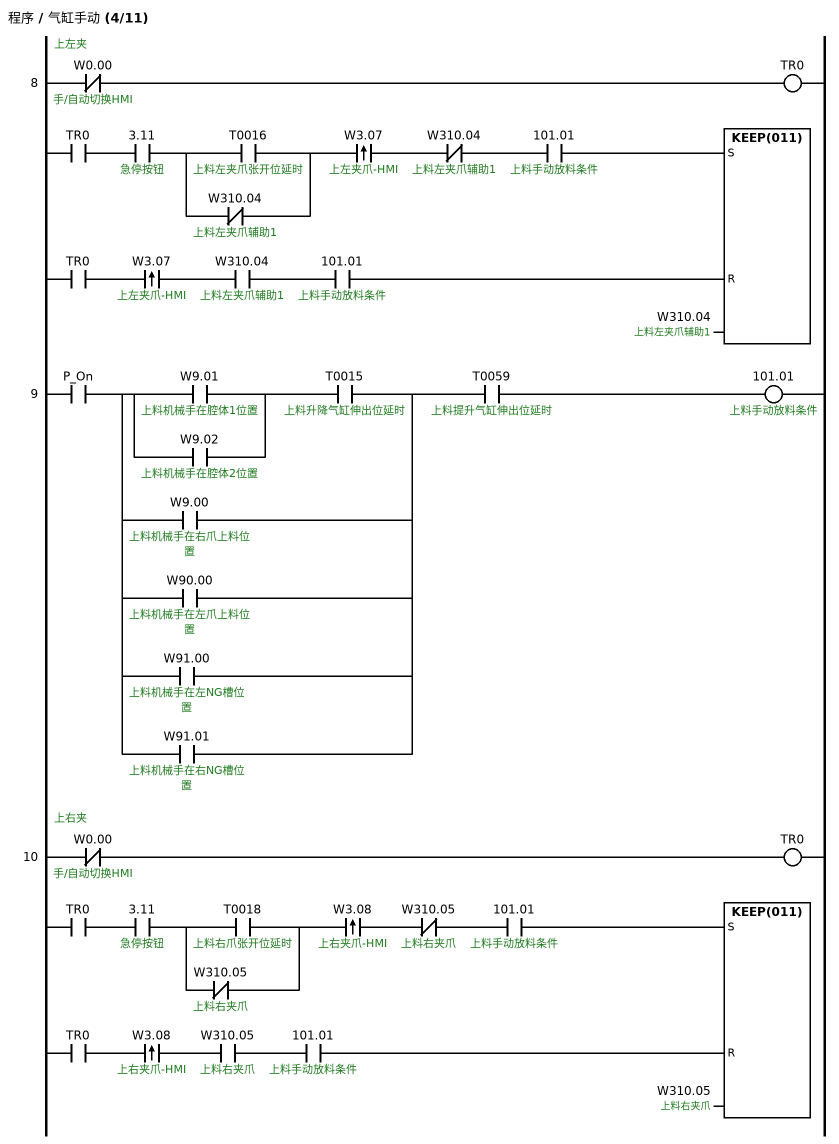
; rung 8: 上左夹
LDNOT W0.00  ; 手/自动切换HMI
OUT TR0
AND 3.11  ; 急停按钮
LD T0016  ; 上料左夹爪张开位延时
ORNOT W310.04  ; 上料左夹爪辅助1
ANDLD
@AND W3.07  ; 上左夹爪-HMI
ANDNOT W310.04  ; 上料左夹爪辅助1
AND 101.01  ; 上料手动放料条件
LD TR0
@AND W3.07  ; 上左夹爪-HMI
AND W310.04  ; 上料左夹爪辅助1
AND 101.01  ; 上料手动放料条件
KEEP(011) W310.04  ; 上料左夹爪辅助1
; rung 9
LD P_On
LD W9.01  ; 上料机械手在腔体1位置
OR W9.02  ; 上料机械手在腔体2位置
AND T0015  ; 上料升降气缸伸出位延时
OR W9.00  ; 上料机械手在右爪上料位置
OR W90.00  ; 上料机械手在左爪上料位置
OR W91.00  ; 上料机械手在左NG槽位置
OR W91.01  ; 上料机械手在右NG槽位置
ANDLD
AND T0059  ; 上料提升气缸伸出位延时
OUT 101.01  ; 上料手动放料条件
; rung 10: 上右夹
LDNOT W0.00  ; 手/自动切换HMI
OUT TR0
AND 3.11  ; 急停按钮
LD T0018  ; 上料右爪张开位延时
ORNOT W310.05  ; 上料右夹爪
ANDLD
@AND W3.08  ; 上右夹爪-HMI
ANDNOT W310.05  ; 上料右夹爪
AND 101.01  ; 上料手动放料条件
LD TR0
@AND W3.08  ; 上右夹爪-HMI
AND W310.05  ; 上料右夹爪
AND 101.01  ; 上料手动放料条件
KEEP(011) W310.05  ; 上料右夹爪

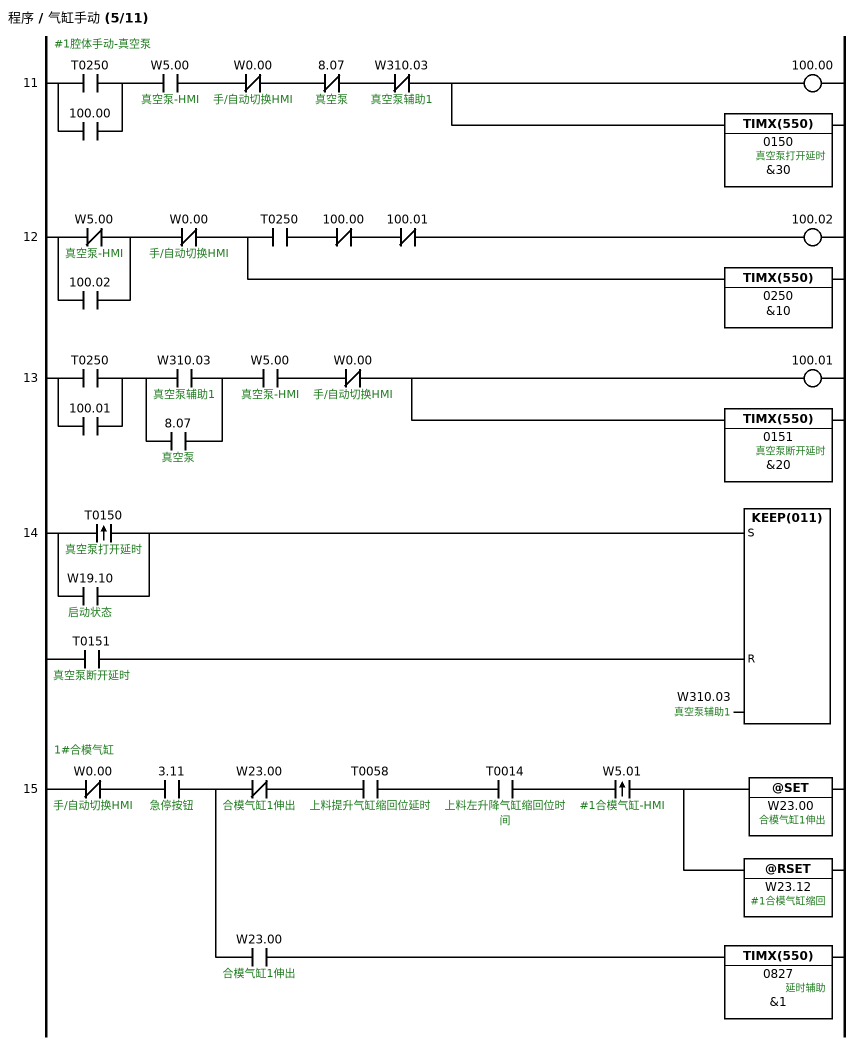
; rung 11: #1腔体手动-真空泵
LD T0250
OR 100.00
AND W5.00  ; 真空泵-HMI
ANDNOT W0.00  ; 手/自动切换HMI
ANDNOT 8.07  ; 真空泵
ANDNOT W310.03  ; 真空泵辅助1
OUT 100.00
TIMX(550) 0150 &30  ; 真空泵打开延时
; rung 12
LDNOT W5.00  ; 真空泵-HMI
OR 100.02
ANDNOT W0.00  ; 手/自动切换HMI
OUT TR0
AND T0250
ANDNOT 100.00
ANDNOT 100.01
OUT 100.02
LD TR0
TIMX(550) 0250 &10
; rung 13
LD T0250
OR 100.01
LD W310.03  ; 真空泵辅助1
OR 8.07  ; 真空泵
ANDLD
AND W5.00  ; 真空泵-HMI
ANDNOT W0.00  ; 手/自动切换HMI
OUT 100.01
TIMX(550) 0151 &20  ; 真空泵断开延时
; rung 14
@LD T0150  ; 真空泵打开延时
OR W19.10  ; 启动状态
LD T0151  ; 真空泵断开延时
KEEP(011) W310.03  ; 真空泵辅助1
; rung 15: 1#合模气缸
LDNOT W0.00  ; 手/自动切换HMI
AND 3.11  ; 急停按钮
OUT TR0
ANDNOT W23.00  ; 合模气缸1伸出
AND T0058  ; 上料提升气缸缩回位延时
AND T0014  ; 上料左升降气缸缩回位时间
@AND W5.01  ; #1合模气缸-HMI
@SET W23.00  ; 合模气缸1伸出
@RSET W23.12  ; #1合模气缸缩回
LD TR0
AND W23.00  ; 合模气缸1伸出
TIMX(550) 0827 &1  ; 延时辅助

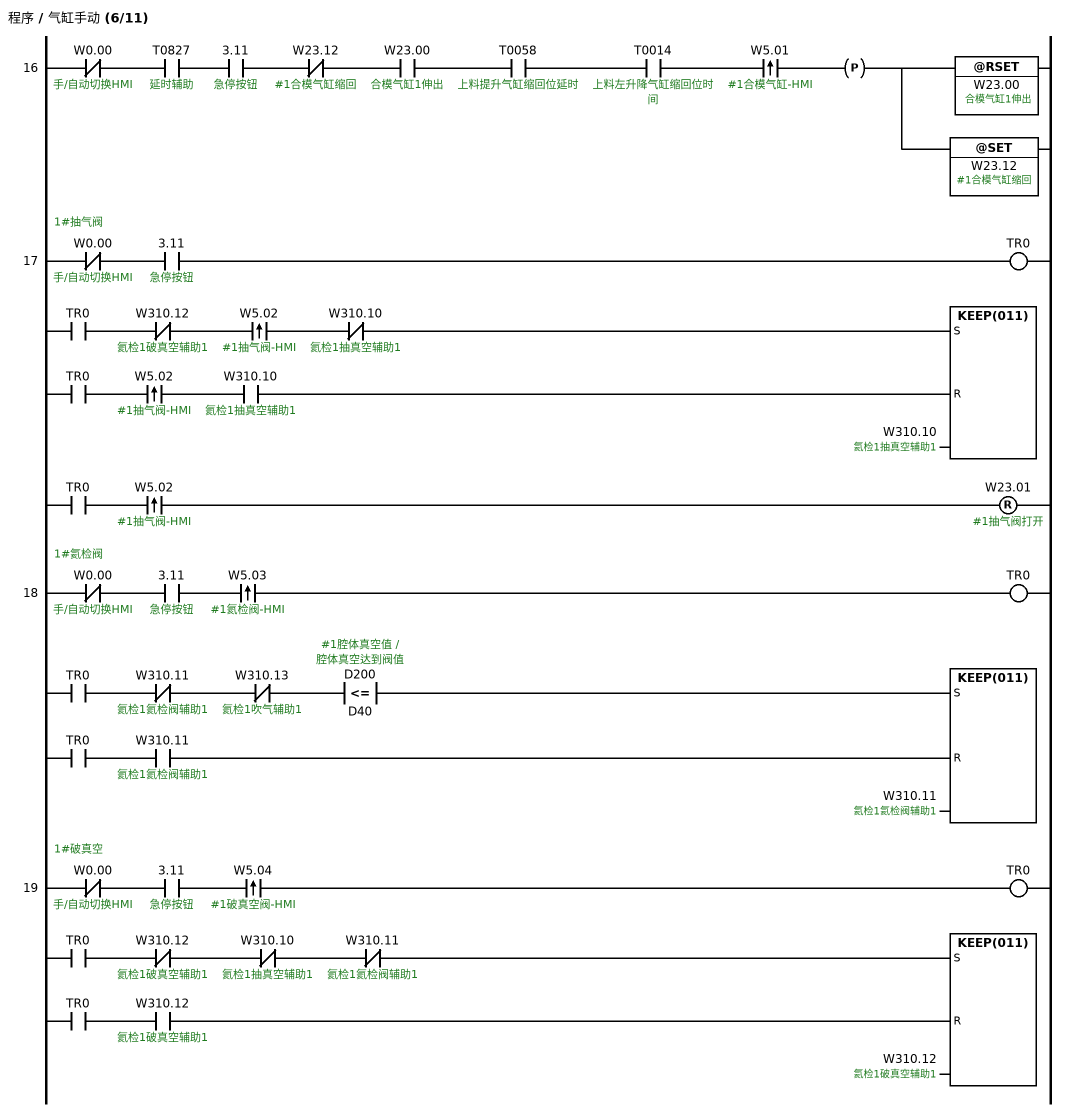
; rung 16
LDNOT W0.00  ; 手/自动切换HMI
AND T0827  ; 延时辅助
AND 3.11  ; 急停按钮
ANDNOT W23.12  ; #1合模气缸缩回
AND W23.00  ; 合模气缸1伸出
AND T0058  ; 上料提升气缸缩回位延时
AND T0014  ; 上料左升降气缸缩回位时间
@AND W5.01  ; #1合模气缸-HMI
UP(521)
@RSET W23.00  ; 合模气缸1伸出
@SET W23.12  ; #1合模气缸缩回
; rung 17: 1#抽气阀
LDNOT W0.00  ; 手/自动切换HMI
AND 3.11  ; 急停按钮
OUT TR0
ANDNOT W310.12  ; 氦检1破真空辅助1
@AND W5.02  ; #1抽气阀-HMI
ANDNOT W310.10  ; 氦检1抽真空辅助1
LD TR0
@AND W5.02  ; #1抽气阀-HMI
AND W310.10  ; 氦检1抽真空辅助1
KEEP(011) W310.10  ; 氦检1抽真空辅助1
LD TR0
@AND W5.02  ; #1抽气阀-HMI
RSET W23.01  ; #1抽气阀打开
; rung 18: 1#氦检阀
LDNOT W0.00  ; 手/自动切换HMI
AND 3.11  ; 急停按钮
@AND W5.03  ; #1氦检阀-HMI
OUT TR0
ANDNOT W310.11  ; 氦检1氦检阀辅助1
ANDNOT W310.13  ; 氦检1吹气辅助1
AND<=F(332) D200 D40  ; #1腔体真空值, 腔体真空达到阀值
LD TR0
AND W310.11  ; 氦检1氦检阀辅助1
KEEP(011) W310.11  ; 氦检1氦检阀辅助1
; rung 19: 1#破真空
LDNOT W0.00  ; 手/自动切换HMI
AND 3.11  ; 急停按钮
@AND W5.04  ; #1破真空阀-HMI
OUT TR0
ANDNOT W310.12  ; 氦检1破真空辅助1
ANDNOT W310.10  ; 氦检1抽真空辅助1
ANDNOT W310.11  ; 氦检1氦检阀辅助1
LD TR0
AND W310.12  ; 氦检1破真空辅助1
KEEP(011) W310.12  ; 氦检1破真空辅助1

